LIN {X -0.154,Y -307.907,Z 608.339,A 0.000,B 0.000,C 90.000,E1 61.051} C_DIS
LIN {X 0.052,Y -298.895,Z 608.321,A 0.000,B 0.000,C 90.000,E1 57.740} C_DIS
LIN {X 0.110,Y -290.449,Z 608.302,A 0.000,B 0.000,C 90.000,E1 54.402} C_DIS
LIN {X -0.081,Y -283.937,Z 608.287,A 0.000,B 0.000,C 90.000,E1 51.743} C_DIS
LIN {X 0.078,Y -278.963,Z 608.276,A 0.000,B 0.000,C 90.000,E1 49.666} C_DIS
LIN {X -0.073,Y -273.546,Z 608.265,A 0.000,B 0.000,C 90.000,E1 47.634} C_DIS
LIN {X 0.074,Y -269.596,Z 608.257,A 0.000,B 0.000,C 90.000,E1 46.215} C_DIS
LIN {X -0.146,Y -264.247,Z 608.247,A 0.000,B 0.000,C 90.000,E1 44.514} C_DIS
LIN {X -0.046,Y -257.475,Z 608.235,A 0.000,B 0.000,C 90.000,E1 42.366} C_DIS
LIN {X -0.013,Y -247.381,Z 608.217,A 0.000,B 0.000,C 90.000,E1 39.116} C_DIS
LIN {X 0.041,Y -238.999,Z 608.201,A 0.000,B 0.000,C 90.000,E1 36.171} C_DIS
LIN {X -0.054,Y -231.454,Z 608.184,A 0.000,B 0.000,C 90.000,E1 33.214} C_DIS
LIN {X -0.001,Y -222.964,Z 608.163,A 0.000,B 0.000,C 90.000,E1 29.411} C_DIS
LIN {X -0.110,Y -217.013,Z 608.146,A 0.000,B 0.000,C 90.000,E1 26.360} C_DIS
LIN {X 0.028,Y -211.815,Z 608.129,A 0.000,B 0.000,C 90.000,E1 23.206} C_DIS
LIN {X 0.001,Y -206.428,Z 608.107,A 0.000,B 0.000,C 90.000,E1 19.268} C_DIS
LIN {X -0.072,Y -202.159,Z 608.085,A 0.000,B 0.000,C 90.000,E1 15.300} C_DIS
LIN {X 0.049,Y -198.456,Z 608.058,A 0.000,B 0.000,C 90.000,E1 10.433} C_DIS
LIN {X -0.013,Y -195.902,Z 608.022,A 0.000,B 0.000,C 90.000,E1 3.955} C_DIS
LIN {X 0.064,Y -197.486,Z 607.961,A 0.000,B 0.000,C 90.000,E1 352.996} C_DIS
LIN {X -0.083,Y -200.607,Z 607.934,A 0.000,B 0.000,C 90.000,E1 348.173} C_DIS
LIN {X -0.002,Y -204.996,Z 607.907,A 0.000,B 0.000,C 90.000,E1 343.323} C_DIS
LIN {X -0.001,Y -209.680,Z 607.885,A 0.000,B 0.000,C 90.000,E1 339.337} C_DIS
LIN {X -0.064,Y -215.034,Z 607.863,A 0.000,B 0.000,C 90.000,E1 335.409} C_DIS
LIN {X -0.075,Y -221.104,Z 607.842,A 0.000,B 0.000,C 90.000,E1 331.513} C_DIS
LIN {X -0.057,Y -227.879,Z 607.820,A 0.000,B 0.000,C 90.000,E1 327.661} C_DIS
LIN {X -0.004,Y -233.659,Z 607.803,A 0.000,B 0.000,C 90.000,E1 324.609} C_DIS
LIN {X -0.099,Y -241.291,Z 607.783,A 0.000,B 0.000,C 90.000,E1 320.884} C_DIS
LIN {X 0.101,Y -249.514,Z 607.762,A 0.000,B 0.000,C 90.000,E1 317.148} C_DIS
LIN {X 0.010,Y -258.785,Z 607.742,A 0.000,B 0.000,C 90.000,E1 313.542} C_DIS
LIN {X 0.036,Y -268.335,Z 607.724,A 0.000,B 0.000,C 90.000,E1 310.334} C_DIS
LIN {X -0.067,Y -280.538,Z 607.705,A 0.000,B 0.000,C 90.000,E1 306.870} C_DIS
LIN {X 0.015,Y -292.771,Z 607.688,A 0.000,B 0.000,C 90.000,E1 303.785} C_DIS
LIN {X 0.005,Y -308.160,Z 607.669,A 0.000,B 0.000,C 90.000,E1 300.463} C_DIS
LIN {X 0.131,Y -321.249,Z 607.655,A 0.000,B 0.000,C 90.000,E1 297.847} C_DIS
LIN {X -0.022,Y -336.716,Z 607.639,A 0.000,B 0.000,C 90.000,E1 295.027} C_DIS
LIN {X -0.066,Y -351.631,Z 607.625,A 0.000,B 0.000,C 90.000,E1 292.567} C_DIS
LIN {X -0.076,Y -369.880,Z 607.610,A 0.000,B 0.000,C 90.000,E1 289.866} C_DIS
LIN {X -0.071,Y -385.394,Z 607.599,A 0.000,B 0.000,C 90.000,E1 287.819} C_DIS
LIN {X 0.169,Y -401.771,Z 607.588,A 0.000,B 0.000,C 90.000,E1 285.788} C_DIS
LIN {X 0.044,Y -413.277,Z 607.580,A 0.000,B 0.000,C 90.000,E1 284.411} C_DIS
LIN {X 0.028,Y -426.894,Z 607.571,A 0.000,B 0.000,C 90.000,E1 282.771} C_DIS
LIN {X -0.124,Y -435.553,Z 607.565,A 0.000,B 0.000,C 90.000,E1 281.715} C_DIS
LIN {X 0.033,Y -445.944,Z 607.558,A 0.000,B 0.000,C 90.000,E1 280.366} C_DIS
LIN {X 0.016,Y -453.769,Z 607.552,A 0.000,B 0.000,C 90.000,E1 279.321} C_DIS
LIN {X 0.090,Y -461.171,Z 607.546,A 0.000,B 0.000,C 90.000,E1 278.276} C_DIS
LIN {X 0.189,Y -468.053,Z 607.540,A 0.000,B 0.000,C 90.000,E1 277.239} C_DIS
LIN {X 0.116,Y -472.817,Z 607.536,A 0.000,B 0.000,C 90.000,E1 276.486} C_DIS
LIN {X 0.025,Y -476.986,Z 607.532,A 0.000,B 0.000,C 90.000,E1 275.739} C_DIS
LIN {X 0.162,Y -479.355,Z 607.529,A 0.000,B 0.000,C 90.000,E1 275.220} C_DIS
LIN {X -0.167,Y -481.369,Z 607.526,A 0.000,B 0.000,C 90.000,E1 274.759} C_DIS
LIN {X -0.049,Y -483.017,Z 607.524,A 0.000,B 0.000,C 90.000,E1 274.245} C_DIS
LIN {X 0.120,Y -484.265,Z 607.521,A 0.000,B 0.000,C 90.000,E1 273.726} C_DIS
LIN {X -0.218,Y -485.178,Z 607.518,A 0.000,B 0.000,C 90.000,E1 273.269} C_DIS
LIN {X -0.035,Y -485.791,Z 607.515,A 0.000,B 0.000,C 90.000,E1 272.751} C_DIS
LIN {X 0.127,Y -486.145,Z 607.513,A 0.000,B 0.000,C 90.000,E1 272.236} C_DIS
LIN {X -0.174,Y -486.217,Z 607.510,A 0.000,B 0.000,C 90.000,E1 271.776} C_DIS
LIN {X -0.004,Y -485.806,Z 607.507,A 0.000,B 0.000,C 90.000,E1 271.260} C_DIS
LIN {X 0.167,Y -485.043,Z 607.504,A 0.000,B 0.000,C 90.000,E1 270.745} C_DIS
LIN {X -0.148,Y -483.736,Z 607.501,A 0.000,B 0.000,C 90.000,E1 270.286} C_DIS
LIN {X 0.018,Y -481.794,Z 607.499,A 0.000,B 0.000,C 90.000,E1 269.771} C_DIS
LIN {X -0.143,Y -480.602,Z 607.497,A 0.000,B 0.000,C 90.000,E1 269.542} C_DIS
LIN {X 0.004,Y -477.592,Z 607.495,A 0.000,B 0.000,C 90.000,E1 269.026} C_DIS
LIN {X 0.131,Y -473.643,Z 607.492,A 0.000,B 0.000,C 90.000,E1 268.511} C_DIS
LIN {X -0.047,Y -471.299,Z 607.490,A 0.000,B 0.000,C 90.000,E1 268.282} C_DIS
LIN {X -0.218,Y -468.627,Z 607.489,A 0.000,B 0.000,C 90.000,E1 268.051} C_DIS
LIN {X 0.063,Y -465.586,Z 607.488,A 0.000,B 0.000,C 90.000,E1 267.764} C_DIS
LIN {X 0.139,Y -462.587,Z 607.486,A 0.000,B 0.000,C 90.000,E1 267.535} C_DIS
LIN {X 0.212,Y -459.159,Z 607.485,A 0.000,B 0.000,C 90.000,E1 267.306} C_DIS
LIN {X 0.043,Y -452.159,Z 607.483,A 0.000,B 0.000,C 90.000,E1 266.963} C_DIS
LIN {X -0.010,Y -444.654,Z 607.482,A 0.000,B 0.000,C 90.000,E1 266.674} C_DIS
LIN {X -0.009,Y -436.831,Z 607.480,A 0.000,B 0.000,C 90.000,E1 266.445} C_DIS
LIN {X -0.012,Y -428.139,Z 607.479,A 0.000,B 0.000,C 90.000,E1 266.274} C_DIS
LIN {X -0.015,Y -418.707,Z 607.479,A 0.000,B 0.000,C 90.000,E1 266.159} C_DIS
LIN {X 0.035,Y -410.839,Z 607.478,A 0.000,B 0.000,C 90.000,E1 266.102} C_DIS
LIN {X -0.016,Y -180.925,Z 607.478,A 0.000,B 0.000,C 90.000,E1 266.102} C_DIS
LIN {X -0.023,Y -180.899,Z 607.474,A 0.000,B 0.000,C 90.000,E1 265.241} C_DIS
LIN {X -0.073,Y -180.214,Z 607.464,A 0.000,B 0.000,C 90.000,E1 263.571} C_DIS
LIN {X 0.057,Y -179.034,Z 607.445,A 0.000,B 0.000,C 90.000,E1 260.151} C_DIS
LIN {X -0.057,Y -178.690,Z 607.441,A 0.000,B 0.000,C 90.000,E1 259.342} C_DIS
LIN {X 0.054,Y -175.740,Z 607.412,A 0.000,B 0.000,C 90.000,E1 254.212} C_DIS
LIN {X 0.049,Y -171.924,Z 607.384,A 0.000,B 0.000,C 90.000,E1 249.082} C_DIS
LIN {X 0.024,Y -171.296,Z 607.379,A 0.000,B 0.000,C 90.000,E1 248.230} C_DIS
LIN {X 0.069,Y -167.560,Z 607.355,A 0.000,B 0.000,C 90.000,E1 243.896} C_DIS
LIN {X 0.082,Y -166.184,Z 607.345,A 0.000,B 0.000,C 90.000,E1 242.153} C_DIS
LIN {X 0.072,Y -162.954,Z 607.326,A 0.000,B 0.000,C 90.000,E1 238.663} C_DIS
LIN {X -0.104,Y -160.862,Z 607.311,A 0.000,B 0.000,C 90.000,E1 236.087} C_DIS
LIN {X 0.096,Y -157.638,Z 607.292,A 0.000,B 0.000,C 90.000,E1 232.477} C_DIS
LIN {X 0.034,Y -155.675,Z 607.277,A 0.000,B 0.000,C 90.000,E1 229.828} C_DIS
LIN {X 0.086,Y -151.941,Z 607.252,A 0.000,B 0.000,C 90.000,E1 225.324} C_DIS
LIN {X 0.100,Y -150.180,Z 607.237,A 0.000,B 0.000,C 90.000,E1 222.609} C_DIS
LIN {X 0.020,Y -146.954,Z 607.212,A 0.000,B 0.000,C 90.000,E1 218.096} C_DIS
LIN {X 0.008,Y -145.541,Z 607.196,A 0.000,B 0.000,C 90.000,E1 215.358} C_DIS
LIN {X -0.075,Y -142.937,Z 607.171,A 0.000,B 0.000,C 90.000,E1 210.797} C_DIS
LIN {X -0.019,Y -141.561,Z 607.150,A 0.000,B 0.000,C 90.000,E1 207.078} C_DIS
LIN {X 0.034,Y -139.409,Z 607.114,A 0.000,B 0.000,C 90.000,E1 200.556} C_DIS
LIN {X -0.044,Y -139.130,Z 607.104,A 0.000,B 0.000,C 90.000,E1 198.725} C_DIS
LIN {X -0.017,Y -138.350,Z 607.057,A 0.000,B 0.000,C 90.000,E1 190.310} C_DIS
LIN {X -0.029,Y -139.498,Z 607.005,A 0.000,B 0.000,C 90.000,E1 180.974} C_DIS
LIN {X 0.052,Y -141.119,Z 606.974,A 0.000,B 0.000,C 90.000,E1 175.355} C_DIS
LIN {X 0.005,Y -142.499,Z 606.959,A 0.000,B 0.000,C 90.000,E1 172.591} C_DIS
LIN {X -0.048,Y -144.754,Z 606.933,A 0.000,B 0.000,C 90.000,E1 167.993} C_DIS
LIN {X 0.043,Y -147.363,Z 606.913,A 0.000,B 0.000,C 90.000,E1 164.283} C_DIS
LIN {X -0.035,Y -150.690,Z 606.887,A 0.000,B 0.000,C 90.000,E1 159.752} C_DIS
LIN {X 0.048,Y -154.170,Z 606.867,A 0.000,B 0.000,C 90.000,E1 156.102} C_DIS
LIN {X -0.022,Y -157.604,Z 606.847,A 0.000,B 0.000,C 90.000,E1 152.538} C_DIS
LIN {X -0.072,Y -161.856,Z 606.828,A 0.000,B 0.000,C 90.000,E1 148.997} C_DIS
LIN {X -0.054,Y -166.047,Z 606.808,A 0.000,B 0.000,C 90.000,E1 145.468} C_DIS
LIN {X -0.063,Y -171.051,Z 606.789,A 0.000,B 0.000,C 90.000,E1 141.984} C_DIS
LIN {X -0.033,Y -175.922,Z 606.770,A 0.000,B 0.000,C 90.000,E1 138.528} C_DIS
LIN {X -0.041,Y -180.161,Z 606.755,A 0.000,B 0.000,C 90.000,E1 135.972} C_DIS
LIN {X -0.072,Y -185.579,Z 606.737,A 0.000,B 0.000,C 90.000,E1 132.609} C_DIS
LIN {X -0.035,Y -191.262,Z 606.719,A 0.000,B 0.000,C 90.000,E1 129.483} C_DIS
LIN {X -0.093,Y -288.943,Z 606.719,A 0.000,B 0.000,C 90.000,E1 129.483} C_DIS
LIN {X -0.106,Y -294.294,Z 606.718,A 0.000,B 0.000,C 90.000,E1 129.277} C_DIS
LIN {X 0.030,Y -297.356,Z 606.717,A 0.000,B 0.000,C 90.000,E1 128.991} C_DIS
LIN {X -0.045,Y -301.065,Z 606.714,A 0.000,B 0.000,C 90.000,E1 128.508} C_DIS
LIN {X -0.051,Y -302.796,Z 606.712,A 0.000,B 0.000,C 90.000,E1 128.177} C_DIS
LIN {X 0.131,Y -304.154,Z 606.710,A 0.000,B 0.000,C 90.000,E1 127.810} C_DIS
LIN {X 0.085,Y -307.941,Z 606.703,A 0.000,B 0.000,C 90.000,E1 126.503} C_DIS
LIN {X -0.122,Y -317.977,Z 606.685,A 0.000,B 0.000,C 90.000,E1 123.293} C_DIS
LIN {X 0.095,Y -328.326,Z 606.669,A 0.000,B 0.000,C 90.000,E1 120.384} C_DIS
LIN {X -0.045,Y -340.030,Z 606.653,A 0.000,B 0.000,C 90.000,E1 117.590} C_DIS
LIN {X -0.003,Y -353.187,Z 606.638,A 0.000,B 0.000,C 90.000,E1 114.823} C_DIS
LIN {X 0.076,Y -366.203,Z 606.625,A 0.000,B 0.000,C 90.000,E1 112.408} C_DIS
LIN {X 0.018,Y -380.557,Z 606.612,A 0.000,B 0.000,C 90.000,E1 110.066} C_DIS
LIN {X 0.054,Y -396.354,Z 606.599,A 0.000,B 0.000,C 90.000,E1 107.764} C_DIS
LIN {X -0.143,Y -413.709,Z 606.586,A 0.000,B 0.000,C 90.000,E1 105.552} C_DIS
LIN {X -0.022,Y -432.735,Z 606.574,A 0.000,B 0.000,C 90.000,E1 103.355} C_DIS
LIN {X 0.049,Y -452.847,Z 606.563,A 0.000,B 0.000,C 90.000,E1 101.299} C_DIS
LIN {X -0.132,Y -473.327,Z 606.552,A 0.000,B 0.000,C 90.000,E1 99.443} C_DIS
LIN {X -0.043,Y -475.167,Z 606.551,A 0.000,B 0.000,C 90.000,E1 99.208} C_DIS
LIN {X -0.182,Y -476.735,Z 606.550,A 0.000,B 0.000,C 90.000,E1 98.973} C_DIS
LIN {X 0.077,Y -477.911,Z 606.548,A 0.000,B 0.000,C 90.000,E1 98.690} C_DIS
LIN {X -0.186,Y -479.333,Z 606.546,A 0.000,B 0.000,C 90.000,E1 98.219} C_DIS
LIN {X -0.038,Y -479.722,Z 606.543,A 0.000,B 0.000,C 90.000,E1 97.701} C_DIS
LIN {X 0.120,Y -479.141,Z 606.540,A 0.000,B 0.000,C 90.000,E1 97.182} C_DIS
LIN {X -0.194,Y -477.502,Z 606.537,A 0.000,B 0.000,C 90.000,E1 96.720} C_DIS
LIN {X 0.149,Y -476.194,Z 606.536,A 0.000,B 0.000,C 90.000,E1 96.429} C_DIS
LIN {X 0.012,Y -465.298,Z 606.527,A 0.000,B 0.000,C 90.000,E1 94.935} C_DIS
LIN {X 0.163,Y -455.064,Z 606.519,A 0.000,B 0.000,C 90.000,E1 93.383} C_DIS
LIN {X 0.069,Y -442.818,Z 606.507,A 0.000,B 0.000,C 90.000,E1 91.318} C_DIS
LIN {X -0.195,Y -434.234,Z 606.499,A 0.000,B 0.000,C 90.000,E1 89.771} C_DIS
LIN {X 0.119,Y -426.716,Z 606.491,A 0.000,B 0.000,C 90.000,E1 88.396} C_DIS
LIN {X 0.033,Y -417.283,Z 606.482,A 0.000,B 0.000,C 90.000,E1 86.788} C_DIS
LIN {X 0.018,Y -403.197,Z 606.468,A 0.000,B 0.000,C 90.000,E1 84.318} C_DIS
LIN {X 0.155,Y -388.249,Z 606.453,A 0.000,B 0.000,C 90.000,E1 81.489} C_DIS
LIN {X -0.001,Y -376.701,Z 606.440,A 0.000,B 0.000,C 90.000,E1 79.218} C_DIS
LIN {X 0.012,Y -365.513,Z 606.427,A 0.000,B 0.000,C 90.000,E1 76.881} C_DIS
LIN {X -0.100,Y -352.191,Z 606.411,A 0.000,B 0.000,C 90.000,E1 73.921} C_DIS
LIN {X 0.021,Y -337.507,Z 606.390,A 0.000,B 0.000,C 90.000,E1 70.242} C_DIS
LIN {X 0.131,Y -325.514,Z 606.371,A 0.000,B 0.000,C 90.000,E1 66.794} C_DIS
LIN {X 0.015,Y -315.551,Z 606.354,A 0.000,B 0.000,C 90.000,E1 63.640} C_DIS
LIN {X 0.068,Y -308.120,Z 606.339,A 0.000,B 0.000,C 90.000,E1 61.051} C_DIS
LIN {X 0.021,Y -299.091,Z 606.321,A 0.000,B 0.000,C 90.000,E1 57.788} C_DIS
LIN {X -0.074,Y -290.637,Z 606.303,A 0.000,B 0.000,C 90.000,E1 54.482} C_DIS
LIN {X -0.036,Y -284.120,Z 606.288,A 0.000,B 0.000,C 90.000,E1 51.778} C_DIS
LIN {X -0.095,Y -279.147,Z 606.276,A 0.000,B 0.000,C 90.000,E1 49.747} C_DIS
LIN {X -0.056,Y -273.737,Z 606.265,A 0.000,B 0.000,C 90.000,E1 47.676} C_DIS
LIN {X -0.089,Y -269.777,Z 606.257,A 0.000,B 0.000,C 90.000,E1 46.296} C_DIS
LIN {X 0.009,Y -265.547,Z 606.249,A 0.000,B 0.000,C 90.000,E1 44.879} C_DIS
LIN {X -0.041,Y -258.820,Z 606.238,A 0.000,B 0.000,C 90.000,E1 42.771} C_DIS
LIN {X 0.015,Y -249.763,Z 606.222,A 0.000,B 0.000,C 90.000,E1 39.886} C_DIS
LIN {X 0.063,Y -239.141,Z 606.201,A 0.000,B 0.000,C 90.000,E1 36.217} C_DIS
LIN {X 0.031,Y -231.589,Z 606.185,A 0.000,B 0.000,C 90.000,E1 33.245} C_DIS
LIN {X 0.080,Y -224.692,Z 606.168,A 0.000,B 0.000,C 90.000,E1 30.207} C_DIS
LIN {X 0.115,Y -218.544,Z 606.151,A 0.000,B 0.000,C 90.000,E1 27.129} C_DIS
LIN {X -0.103,Y -213.122,Z 606.134,A 0.000,B 0.000,C 90.000,E1 24.079} C_DIS
LIN {X -0.011,Y -207.491,Z 606.112,A 0.000,B 0.000,C 90.000,E1 20.120} C_DIS
LIN {X 0.009,Y -202.956,Z 606.090,A 0.000,B 0.000,C 90.000,E1 16.134} C_DIS
LIN {X 0.047,Y -199.020,Z 606.063,A 0.000,B 0.000,C 90.000,E1 11.299} C_DIS
LIN {X 0.036,Y -196.308,Z 606.031,A 0.000,B 0.000,C 90.000,E1 5.625} C_DIS
LIN {X 0.064,Y -197.506,Z 605.961,A 0.000,B 0.000,C 90.000,E1 352.996} C_DIS
LIN {X -0.081,Y -200.649,Z 605.934,A 0.000,B 0.000,C 90.000,E1 348.173} C_DIS
LIN {X 0.000,Y -205.029,Z 605.907,A 0.000,B 0.000,C 90.000,E1 343.323} C_DIS
LIN {X 0.003,Y -209.708,Z 605.885,A 0.000,B 0.000,C 90.000,E1 339.337} C_DIS
LIN {X -0.059,Y -215.060,Z 605.863,A 0.000,B 0.000,C 90.000,E1 335.409} C_DIS
LIN {X -0.068,Y -221.137,Z 605.842,A 0.000,B 0.000,C 90.000,E1 331.513} C_DIS
LIN {X -0.050,Y -227.896,Z 605.820,A 0.000,B 0.000,C 90.000,E1 327.661} C_DIS
LIN {X -0.030,Y -235.138,Z 605.799,A 0.000,B 0.000,C 90.000,E1 323.863} C_DIS
LIN {X 0.025,Y -242.853,Z 605.778,A 0.000,B 0.000,C 90.000,E1 320.114} C_DIS
LIN {X -0.070,Y -251.235,Z 605.758,A 0.000,B 0.000,C 90.000,E1 316.458} C_DIS
LIN {X -0.111,Y -260.744,Z 605.738,A 0.000,B 0.000,C 90.000,E1 312.852} C_DIS
LIN {X -0.023,Y -270.590,Z 605.720,A 0.000,B 0.000,C 90.000,E1 309.644} C_DIS
LIN {X -0.007,Y -283.114,Z 605.701,A 0.000,B 0.000,C 90.000,E1 306.171} C_DIS
LIN {X 0.019,Y -292.723,Z 605.688,A 0.000,B 0.000,C 90.000,E1 303.785} C_DIS
LIN {X 0.005,Y -308.088,Z 605.669,A 0.000,B 0.000,C 90.000,E1 300.463} C_DIS
LIN {X 0.129,Y -321.151,Z 605.655,A 0.000,B 0.000,C 90.000,E1 297.847} C_DIS
LIN {X -0.051,Y -338.391,Z 605.637,A 0.000,B 0.000,C 90.000,E1 294.719} C_DIS
LIN {X -0.016,Y -355.459,Z 605.622,A 0.000,B 0.000,C 90.000,E1 291.950} C_DIS
LIN {X -0.126,Y -371.969,Z 605.609,A 0.000,B 0.000,C 90.000,E1 289.577} C_DIS
LIN {X -0.076,Y -397.069,Z 605.591,A 0.000,B 0.000,C 90.000,E1 286.386} C_DIS
LIN {X 0.121,Y -408.725,Z 605.583,A 0.000,B 0.000,C 90.000,E1 284.954} C_DIS
LIN {X -0.135,Y -424.690,Z 605.572,A 0.000,B 0.000,C 90.000,E1 283.063} C_DIS
LIN {X 0.106,Y -433.465,Z 605.566,A 0.000,B 0.000,C 90.000,E1 281.951} C_DIS
LIN {X -0.189,Y -443.962,Z 605.559,A 0.000,B 0.000,C 90.000,E1 280.658} C_DIS
LIN {X 0.213,Y -451.909,Z 605.553,A 0.000,B 0.000,C 90.000,E1 279.557} C_DIS
LIN {X -0.183,Y -459.380,Z 605.547,A 0.000,B 0.000,C 90.000,E1 278.568} C_DIS
LIN {X -0.109,Y -466.347,Z 605.542,A 0.000,B 0.000,C 90.000,E1 277.530} C_DIS
LIN {X 0.111,Y -472.755,Z 605.536,A 0.000,B 0.000,C 90.000,E1 276.486} C_DIS
LIN {X 0.019,Y -476.899,Z 605.532,A 0.000,B 0.000,C 90.000,E1 275.739} C_DIS
LIN {X 0.155,Y -479.288,Z 605.529,A 0.000,B 0.000,C 90.000,E1 275.220} C_DIS
LIN {X -0.174,Y -481.306,Z 605.526,A 0.000,B 0.000,C 90.000,E1 274.759} C_DIS
LIN {X -0.056,Y -482.966,Z 605.524,A 0.000,B 0.000,C 90.000,E1 274.245} C_DIS
LIN {X 0.112,Y -484.232,Z 605.521,A 0.000,B 0.000,C 90.000,E1 273.726} C_DIS
LIN {X -0.225,Y -485.166,Z 605.518,A 0.000,B 0.000,C 90.000,E1 273.269} C_DIS
LIN {X -0.044,Y -485.815,Z 605.515,A 0.000,B 0.000,C 90.000,E1 272.751} C_DIS
LIN {X 0.120,Y -486.126,Z 605.513,A 0.000,B 0.000,C 90.000,E1 272.236} C_DIS
LIN {X -0.182,Y -486.172,Z 605.510,A 0.000,B 0.000,C 90.000,E1 271.776} C_DIS
LIN {X -0.013,Y -485.880,Z 605.507,A 0.000,B 0.000,C 90.000,E1 271.260} C_DIS
LIN {X 0.159,Y -485.075,Z 605.504,A 0.000,B 0.000,C 90.000,E1 270.745} C_DIS
LIN {X -0.156,Y -483.746,Z 605.501,A 0.000,B 0.000,C 90.000,E1 270.286} C_DIS
LIN {X 0.010,Y -481.874,Z 605.499,A 0.000,B 0.000,C 90.000,E1 269.771} C_DIS
LIN {X 0.167,Y -479.239,Z 605.496,A 0.000,B 0.000,C 90.000,E1 269.255} C_DIS
LIN {X -0.173,Y -475.770,Z 605.493,A 0.000,B 0.000,C 90.000,E1 268.797} C_DIS
LIN {X -0.054,Y -471.288,Z 605.490,A 0.000,B 0.000,C 90.000,E1 268.282} C_DIS
LIN {X -0.225,Y -468.587,Z 605.489,A 0.000,B 0.000,C 90.000,E1 268.051} C_DIS
LIN {X 0.056,Y -465.563,Z 605.488,A 0.000,B 0.000,C 90.000,E1 267.764} C_DIS
LIN {X 0.125,Y -462.549,Z 605.486,A 0.000,B 0.000,C 90.000,E1 267.535} C_DIS
LIN {X 0.192,Y -459.093,Z 605.485,A 0.000,B 0.000,C 90.000,E1 267.306} C_DIS
LIN {X 0.031,Y -452.126,Z 605.483,A 0.000,B 0.000,C 90.000,E1 266.963} C_DIS
LIN {X -0.034,Y -444.549,Z 605.482,A 0.000,B 0.000,C 90.000,E1 266.674} C_DIS
LIN {X -0.010,Y -436.839,Z 605.480,A 0.000,B 0.000,C 90.000,E1 266.445} C_DIS
LIN {X 0.003,Y -428.221,Z 605.479,A 0.000,B 0.000,C 90.000,E1 266.274} C_DIS
LIN {X 0.001,Y -418.631,Z 605.479,A 0.000,B 0.000,C 90.000,E1 266.159} C_DIS
LIN {X 0.053,Y -411.194,Z 605.478,A 0.000,B 0.000,C 90.000,E1 266.102} C_DIS
LIN {X -0.020,Y -405.738,Z 605.478,A 0.000,B 0.000,C 90.000,E1 266.102} C_DIS
LIN {X -0.040,Y -180.924,Z 605.478,A 0.000,B 0.000,C 90.000,E1 266.102} C_DIS
LIN {X 0.004,Y -180.875,Z 605.473,A 0.000,B 0.000,C 90.000,E1 265.065} C_DIS
LIN {X 0.087,Y -178.942,Z 605.443,A 0.000,B 0.000,C 90.000,E1 259.803} C_DIS
LIN {X -0.046,Y -175.992,Z 605.415,A 0.000,B 0.000,C 90.000,E1 254.755} C_DIS
LIN {X 0.069,Y -175.495,Z 605.410,A 0.000,B 0.000,C 90.000,E1 253.866} C_DIS
LIN {X -0.037,Y -172.238,Z 605.387,A 0.000,B 0.000,C 90.000,E1 249.625} C_DIS
LIN {X -0.058,Y -171.715,Z 605.382,A 0.000,B 0.000,C 90.000,E1 248.773} C_DIS
LIN {X 0.026,Y -167.311,Z 605.353,A 0.000,B 0.000,C 90.000,E1 243.563} C_DIS
LIN {X 0.032,Y -166.691,Z 605.348,A 0.000,B 0.000,C 90.000,E1 242.692} C_DIS
LIN {X 0.023,Y -162.673,Z 605.324,A 0.000,B 0.000,C 90.000,E1 238.329} C_DIS
LIN {X -0.004,Y -161.362,Z 605.314,A 0.000,B 0.000,C 90.000,E1 236.580} C_DIS
LIN {X 0.030,Y -157.356,Z 605.290,A 0.000,B 0.000,C 90.000,E1 232.145} C_DIS
LIN {X 0.058,Y -155.345,Z 605.275,A 0.000,B 0.000,C 90.000,E1 229.461} C_DIS
LIN {X -0.012,Y -151.692,Z 605.250,A 0.000,B 0.000,C 90.000,E1 225.000} C_DIS
LIN {X 0.036,Y -150.554,Z 605.240,A 0.000,B 0.000,C 90.000,E1 223.176} C_DIS
LIN {X -0.047,Y -147.281,Z 605.215,A 0.000,B 0.000,C 90.000,E1 218.669} C_DIS
LIN {X 0.040,Y -145.309,Z 605.194,A 0.000,B 0.000,C 90.000,E1 214.978} C_DIS
LIN {X 0.032,Y -142.399,Z 605.164,A 0.000,B 0.000,C 90.000,E1 209.461} C_DIS
LIN {X 0.015,Y -141.382,Z 605.148,A 0.000,B 0.000,C 90.000,E1 206.693} C_DIS
LIN {X 0.056,Y -139.349,Z 605.112,A 0.000,B 0.000,C 90.000,E1 200.174} C_DIS
LIN {X -0.002,Y -138.787,Z 605.097,A 0.000,B 0.000,C 90.000,E1 197.402} C_DIS
LIN {X 0.056,Y -138.344,Z 605.055,A 0.000,B 0.000,C 90.000,E1 189.905} C_DIS
LIN {X -0.063,Y -139.386,Z 605.008,A 0.000,B 0.000,C 90.000,E1 181.547} C_DIS
LIN {X -0.010,Y -141.283,Z 604.972,A 0.000,B 0.000,C 90.000,E1 175.008} C_DIS
LIN {X -0.052,Y -142.646,Z 604.957,A 0.000,B 0.000,C 90.000,E1 172.243} C_DIS
LIN {X 0.039,Y -144.982,Z 604.931,A 0.000,B 0.000,C 90.000,E1 167.589} C_DIS
LIN {X 0.030,Y -147.610,Z 604.911,A 0.000,B 0.000,C 90.000,E1 163.921} C_DIS
LIN {X -0.032,Y -150.232,Z 604.890,A 0.000,B 0.000,C 90.000,E1 160.296} C_DIS
LIN {X -0.017,Y -153.623,Z 604.870,A 0.000,B 0.000,C 90.000,E1 156.666} C_DIS
LIN {X -0.029,Y -157.040,Z 604.850,A 0.000,B 0.000,C 90.000,E1 153.076} C_DIS
LIN {X 0.040,Y -161.165,Z 604.831,A 0.000,B 0.000,C 90.000,E1 149.488} C_DIS
LIN {X -0.016,Y -163.261,Z 604.821,A 0.000,B 0.000,C 90.000,E1 147.740} C_DIS
LIN {X 0.082,Y -167.699,Z 604.801,A 0.000,B 0.000,C 90.000,E1 144.196} C_DIS
LIN {X -0.005,Y -171.520,Z 604.787,A 0.000,B 0.000,C 90.000,E1 141.618} C_DIS
LIN {X 0.038,Y -176.458,Z 604.768,A 0.000,B 0.000,C 90.000,E1 138.162} C_DIS
LIN {X -0.091,Y -180.754,Z 604.753,A 0.000,B 0.000,C 90.000,E1 135.648} C_DIS
LIN {X 0.027,Y -186.159,Z 604.735,A 0.000,B 0.000,C 90.000,E1 132.243} C_DIS
LIN {X -0.052,Y -191.271,Z 604.719,A 0.000,B 0.000,C 90.000,E1 129.483} C_DIS
LIN {X -0.114,Y -288.437,Z 604.719,A 0.000,B 0.000,C 90.000,E1 129.483} C_DIS
LIN {X 0.031,Y -291.041,Z 604.719,A 0.000,B 0.000,C 90.000,E1 129.402} C_DIS
LIN {X -0.154,Y -295.400,Z 604.718,A 0.000,B 0.000,C 90.000,E1 129.197} C_DIS
LIN {X 0.078,Y -297.932,Z 604.716,A 0.000,B 0.000,C 90.000,E1 128.910} C_DIS
LIN {X -0.022,Y -301.701,Z 604.713,A 0.000,B 0.000,C 90.000,E1 128.382} C_DIS
LIN {X 0.161,Y -303.293,Z 604.711,A 0.000,B 0.000,C 90.000,E1 128.016} C_DIS
LIN {X -0.081,Y -304.544,Z 604.710,A 0.000,B 0.000,C 90.000,E1 127.729} C_DIS
LIN {X 0.066,Y -316.213,Z 604.688,A 0.000,B 0.000,C 90.000,E1 123.785} C_DIS
LIN {X -0.035,Y -326.327,Z 604.672,A 0.000,B 0.000,C 90.000,E1 120.924} C_DIS
LIN {X -0.072,Y -337.778,Z 604.656,A 0.000,B 0.000,C 90.000,E1 118.103} C_DIS
LIN {X -0.098,Y -350.662,Z 604.641,A 0.000,B 0.000,C 90.000,E1 115.335} C_DIS
LIN {X 0.058,Y -363.416,Z 604.627,A 0.000,B 0.000,C 90.000,E1 112.898} C_DIS
LIN {X -0.075,Y -377.489,Z 604.614,A 0.000,B 0.000,C 90.000,E1 110.556} C_DIS
LIN {X 0.005,Y -392.981,Z 604.601,A 0.000,B 0.000,C 90.000,E1 108.236} C_DIS
LIN {X 0.110,Y -410.008,Z 604.589,A 0.000,B 0.000,C 90.000,E1 105.969} C_DIS
LIN {X 0.141,Y -428.692,Z 604.577,A 0.000,B 0.000,C 90.000,E1 103.772} C_DIS
LIN {X -0.049,Y -448.669,Z 604.565,A 0.000,B 0.000,C 90.000,E1 101.715} C_DIS
LIN {X 0.043,Y -469.223,Z 604.554,A 0.000,B 0.000,C 90.000,E1 99.792} C_DIS
LIN {X 0.100,Y -471.843,Z 604.553,A 0.000,B 0.000,C 90.000,E1 99.557} C_DIS
LIN {X 0.196,Y -474.068,Z 604.552,A 0.000,B 0.000,C 90.000,E1 99.321} C_DIS
LIN {X -0.253,Y -475.755,Z 604.551,A 0.000,B 0.000,C 90.000,E1 99.151} C_DIS
LIN {X 0.080,Y -477.205,Z 604.549,A 0.000,B 0.000,C 90.000,E1 98.859} C_DIS
LIN {X -0.057,Y -478.285,Z 604.548,A 0.000,B 0.000,C 90.000,E1 98.624} C_DIS
LIN {X 0.086,Y -479.555,Z 604.545,A 0.000,B 0.000,C 90.000,E1 98.106} C_DIS
LIN {X -0.238,Y -479.811,Z 604.542,A 0.000,B 0.000,C 90.000,E1 97.644} C_DIS
LIN {X -0.078,Y -479.095,Z 604.540,A 0.000,B 0.000,C 90.000,E1 97.125} C_DIS
LIN {X 0.083,Y -477.291,Z 604.537,A 0.000,B 0.000,C 90.000,E1 96.606} C_DIS
LIN {X -0.048,Y -475.875,Z 604.535,A 0.000,B 0.000,C 90.000,E1 96.372} C_DIS
LIN {X 0.146,Y -459.619,Z 604.523,A 0.000,B 0.000,C 90.000,E1 94.073} C_DIS
LIN {X 0.162,Y -446.885,Z 604.511,A 0.000,B 0.000,C 90.000,E1 92.007} C_DIS
LIN {X -0.125,Y -435.320,Z 604.500,A 0.000,B 0.000,C 90.000,E1 89.943} C_DIS
LIN {X 0.202,Y -427.861,Z 604.492,A 0.000,B 0.000,C 90.000,E1 88.568} C_DIS
LIN {X 0.111,Y -418.438,Z 604.483,A 0.000,B 0.000,C 90.000,E1 86.963} C_DIS
LIN {X 0.154,Y -404.322,Z 604.469,A 0.000,B 0.000,C 90.000,E1 84.489} C_DIS
LIN {X -0.115,Y -389.328,Z 604.454,A 0.000,B 0.000,C 90.000,E1 81.724} C_DIS
LIN {X 0.144,Y -376.306,Z 604.440,A 0.000,B 0.000,C 90.000,E1 79.106} C_DIS
LIN {X 0.137,Y -365.118,Z 604.427,A 0.000,B 0.000,C 90.000,E1 76.769} C_DIS
LIN {X 0.035,Y -350.543,Z 604.408,A 0.000,B 0.000,C 90.000,E1 73.504} C_DIS
LIN {X 0.087,Y -336.050,Z 604.388,A 0.000,B 0.000,C 90.000,E1 69.826} C_DIS
LIN {X -0.074,Y -323.207,Z 604.367,A 0.000,B 0.000,C 90.000,E1 66.102} C_DIS
LIN {X 0.168,Y -313.460,Z 604.349,A 0.000,B 0.000,C 90.000,E1 62.871} C_DIS
LIN {X -0.105,Y -306.068,Z 604.335,A 0.000,B 0.000,C 90.000,E1 60.333} C_DIS
LIN {X -0.056,Y -297.174,Z 604.317,A 0.000,B 0.000,C 90.000,E1 57.041} C_DIS
LIN {X 0.050,Y -290.463,Z 604.302,A 0.000,B 0.000,C 90.000,E1 54.356} C_DIS
LIN {X 0.028,Y -283.942,Z 604.287,A 0.000,B 0.000,C 90.000,E1 51.662} C_DIS
LIN {X 0.006,Y -278.952,Z 604.276,A 0.000,B 0.000,C 90.000,E1 49.622} C_DIS
LIN {X 0.035,Y -275.379,Z 604.268,A 0.000,B 0.000,C 90.000,E1 48.243} C_DIS
LIN {X 0.019,Y -271.537,Z 604.260,A 0.000,B 0.000,C 90.000,E1 46.863} C_DIS
LIN {X -0.053,Y -267.416,Z 604.253,A 0.000,B 0.000,C 90.000,E1 45.486} C_DIS
LIN {X 0.064,Y -261.905,Z 604.243,A 0.000,B 0.000,C 90.000,E1 43.704} C_DIS
LIN {X 0.001,Y -252.812,Z 604.227,A 0.000,B 0.000,C 90.000,E1 40.862} C_DIS
LIN {X -0.052,Y -242.975,Z 604.209,A 0.000,B 0.000,C 90.000,E1 37.604} C_DIS
LIN {X 0.093,Y -234.981,Z 604.192,A 0.000,B 0.000,C 90.000,E1 34.612} C_DIS
LIN {X -0.013,Y -226.101,Z 604.172,A 0.000,B 0.000,C 90.000,E1 30.875} C_DIS
LIN {X -0.132,Y -219.775,Z 604.155,A 0.000,B 0.000,C 90.000,E1 27.847} C_DIS
LIN {X -0.025,Y -214.201,Z 604.137,A 0.000,B 0.000,C 90.000,E1 24.719} C_DIS
LIN {X -0.045,Y -209.443,Z 604.120,A 0.000,B 0.000,C 90.000,E1 21.589} C_DIS
LIN {X -0.091,Y -204.485,Z 604.098,A 0.000,B 0.000,C 90.000,E1 17.638} C_DIS
LIN {X 0.055,Y -200.708,Z 604.076,A 0.000,B 0.000,C 90.000,E1 13.592} C_DIS
LIN {X 0.049,Y -197.487,Z 604.049,A 0.000,B 0.000,C 90.000,E1 8.746} C_DIS
LIN {X 0.049,Y -198.424,Z 603.952,A 0.000,B 0.000,C 90.000,E1 351.376} C_DIS
LIN {X 0.013,Y -202.029,Z 603.925,A 0.000,B 0.000,C 90.000,E1 346.533} C_DIS
LIN {X -0.070,Y -205.948,Z 603.903,A 0.000,B 0.000,C 90.000,E1 342.543} C_DIS
LIN {X 0.028,Y -210.754,Z 603.881,A 0.000,B 0.000,C 90.000,E1 338.539} C_DIS
LIN {X 0.087,Y -216.241,Z 603.859,A 0.000,B 0.000,C 90.000,E1 334.588} C_DIS
LIN {X 0.025,Y -222.452,Z 603.837,A 0.000,B 0.000,C 90.000,E1 330.717} C_DIS
LIN {X -0.107,Y -229.330,Z 603.816,A 0.000,B 0.000,C 90.000,E1 326.914} C_DIS
LIN {X -0.100,Y -236.619,Z 603.795,A 0.000,B 0.000,C 90.000,E1 323.130} C_DIS
LIN {X 0.006,Y -244.429,Z 603.774,A 0.000,B 0.000,C 90.000,E1 319.380} C_DIS
LIN {X -0.058,Y -252.996,Z 603.754,A 0.000,B 0.000,C 90.000,E1 315.729} C_DIS
LIN {X -0.037,Y -262.758,Z 603.734,A 0.000,B 0.000,C 90.000,E1 312.123} C_DIS
LIN {X 0.057,Y -271.704,Z 603.718,A 0.000,B 0.000,C 90.000,E1 309.277} C_DIS
LIN {X 0.115,Y -284.386,Z 603.699,A 0.000,B 0.000,C 90.000,E1 305.804} C_DIS
LIN {X 0.008,Y -294.128,Z 603.686,A 0.000,B 0.000,C 90.000,E1 303.452} C_DIS
LIN {X 0.043,Y -309.612,Z 603.667,A 0.000,B 0.000,C 90.000,E1 300.129} C_DIS
LIN {X -0.152,Y -324.412,Z 603.651,A 0.000,B 0.000,C 90.000,E1 297.257} C_DIS
LIN {X 0.059,Y -341.947,Z 603.634,A 0.000,B 0.000,C 90.000,E1 294.079} C_DIS
LIN {X -0.072,Y -359.392,Z 603.619,A 0.000,B 0.000,C 90.000,E1 291.354} C_DIS
LIN {X -0.049,Y -374.104,Z 603.607,A 0.000,B 0.000,C 90.000,E1 289.268} C_DIS
LIN {X -0.089,Y -397.084,Z 603.591,A 0.000,B 0.000,C 90.000,E1 286.386} C_DIS
LIN {X 0.108,Y -408.699,Z 603.583,A 0.000,B 0.000,C 90.000,E1 284.954} C_DIS
LIN {X 0.112,Y -422.447,Z 603.574,A 0.000,B 0.000,C 90.000,E1 283.300} C_DIS
LIN {X -0.090,Y -431.352,Z 603.568,A 0.000,B 0.000,C 90.000,E1 282.243} C_DIS
LIN {X 0.008,Y -441.994,Z 603.561,A 0.000,B 0.000,C 90.000,E1 280.894} C_DIS
LIN {X -0.054,Y -450.044,Z 603.555,A 0.000,B 0.000,C 90.000,E1 279.849} C_DIS
LIN {X -0.205,Y -459.418,Z 603.547,A 0.000,B 0.000,C 90.000,E1 278.568} C_DIS
LIN {X -0.129,Y -466.350,Z 603.542,A 0.000,B 0.000,C 90.000,E1 277.530} C_DIS
LIN {X 0.089,Y -472.720,Z 603.536,A 0.000,B 0.000,C 90.000,E1 276.486} C_DIS
LIN {X -0.003,Y -476.856,Z 603.532,A 0.000,B 0.000,C 90.000,E1 275.739} C_DIS
LIN {X -0.052,Y -480.281,Z 603.528,A 0.000,B 0.000,C 90.000,E1 274.992} C_DIS
LIN {X -0.197,Y -481.280,Z 603.526,A 0.000,B 0.000,C 90.000,E1 274.759} C_DIS
LIN {X -0.073,Y -482.929,Z 603.524,A 0.000,B 0.000,C 90.000,E1 274.245} C_DIS
LIN {X 0.095,Y -484.197,Z 603.521,A 0.000,B 0.000,C 90.000,E1 273.726} C_DIS
LIN {X -0.243,Y -485.141,Z 603.518,A 0.000,B 0.000,C 90.000,E1 273.269} C_DIS
LIN {X -0.062,Y -485.826,Z 603.515,A 0.000,B 0.000,C 90.000,E1 272.751} C_DIS
LIN {X 0.101,Y -486.168,Z 603.513,A 0.000,B 0.000,C 90.000,E1 272.236} C_DIS
LIN {X -0.200,Y -486.232,Z 603.510,A 0.000,B 0.000,C 90.000,E1 271.776} C_DIS
LIN {X -0.030,Y -485.939,Z 603.507,A 0.000,B 0.000,C 90.000,E1 271.260} C_DIS
LIN {X 0.142,Y -485.116,Z 603.504,A 0.000,B 0.000,C 90.000,E1 270.745} C_DIS
LIN {X -0.172,Y -483.814,Z 603.501,A 0.000,B 0.000,C 90.000,E1 270.286} C_DIS
LIN {X -0.006,Y -481.893,Z 603.499,A 0.000,B 0.000,C 90.000,E1 269.771} C_DIS
LIN {X 0.151,Y -479.265,Z 603.496,A 0.000,B 0.000,C 90.000,E1 269.255} C_DIS
LIN {X -0.189,Y -475.785,Z 603.493,A 0.000,B 0.000,C 90.000,E1 268.797} C_DIS
LIN {X 0.108,Y -473.674,Z 603.492,A 0.000,B 0.000,C 90.000,E1 268.511} C_DIS
LIN {X 0.232,Y -468.586,Z 603.489,A 0.000,B 0.000,C 90.000,E1 267.993} C_DIS
LIN {X 0.049,Y -465.556,Z 603.488,A 0.000,B 0.000,C 90.000,E1 267.764} C_DIS
LIN {X 0.194,Y -459.106,Z 603.485,A 0.000,B 0.000,C 90.000,E1 267.306} C_DIS
LIN {X 0.003,Y -452.041,Z 603.483,A 0.000,B 0.000,C 90.000,E1 266.963} C_DIS
LIN {X -0.066,Y -444.444,Z 603.481,A 0.000,B 0.000,C 90.000,E1 266.674} C_DIS
LIN {X -0.038,Y -436.727,Z 603.480,A 0.000,B 0.000,C 90.000,E1 266.445} C_DIS
LIN {X -0.017,Y -428.020,Z 603.479,A 0.000,B 0.000,C 90.000,E1 266.274} C_DIS
LIN {X -0.005,Y -418.362,Z 603.479,A 0.000,B 0.000,C 90.000,E1 266.159} C_DIS
LIN {X 0.049,Y -410.822,Z 603.478,A 0.000,B 0.000,C 90.000,E1 266.102} C_DIS
LIN {X -0.010,Y -180.924,Z 603.478,A 0.000,B 0.000,C 90.000,E1 266.102} C_DIS
LIN {X -0.015,Y -180.899,Z 603.474,A 0.000,B 0.000,C 90.000,E1 265.241} C_DIS
LIN {X -0.065,Y -180.216,Z 603.464,A 0.000,B 0.000,C 90.000,E1 263.571} C_DIS
LIN {X 0.065,Y -179.034,Z 603.445,A 0.000,B 0.000,C 90.000,E1 260.151} C_DIS
LIN {X -0.049,Y -178.692,Z 603.441,A 0.000,B 0.000,C 90.000,E1 259.342} C_DIS
LIN {X 0.062,Y -175.741,Z 603.412,A 0.000,B 0.000,C 90.000,E1 254.212} C_DIS
LIN {X 0.057,Y -171.925,Z 603.384,A 0.000,B 0.000,C 90.000,E1 249.082} C_DIS
LIN {X 0.031,Y -171.299,Z 603.379,A 0.000,B 0.000,C 90.000,E1 248.230} C_DIS
LIN {X 0.077,Y -167.562,Z 603.355,A 0.000,B 0.000,C 90.000,E1 243.896} C_DIS
LIN {X 0.090,Y -166.187,Z 603.345,A 0.000,B 0.000,C 90.000,E1 242.153} C_DIS
LIN {X 0.080,Y -162.956,Z 603.326,A 0.000,B 0.000,C 90.000,E1 238.663} C_DIS
LIN {X -0.096,Y -160.865,Z 603.311,A 0.000,B 0.000,C 90.000,E1 236.087} C_DIS
LIN {X 0.008,Y -157.639,Z 603.292,A 0.000,B 0.000,C 90.000,E1 232.512} C_DIS
LIN {X 0.041,Y -155.677,Z 603.277,A 0.000,B 0.000,C 90.000,E1 229.828} C_DIS
LIN {X -0.013,Y -151.943,Z 603.252,A 0.000,B 0.000,C 90.000,E1 225.364} C_DIS
LIN {X -0.003,Y -150.182,Z 603.237,A 0.000,B 0.000,C 90.000,E1 222.651} C_DIS
LIN {X 0.027,Y -146.955,Z 603.212,A 0.000,B 0.000,C 90.000,E1 218.096} C_DIS
LIN {X -0.070,Y -145.543,Z 603.196,A 0.000,B 0.000,C 90.000,E1 215.391} C_DIS
LIN {X -0.069,Y -142.938,Z 603.171,A 0.000,B 0.000,C 90.000,E1 210.797} C_DIS
LIN {X -0.011,Y -141.563,Z 603.150,A 0.000,B 0.000,C 90.000,E1 207.078} C_DIS
LIN {X 0.041,Y -139.410,Z 603.114,A 0.000,B 0.000,C 90.000,E1 200.556} C_DIS
LIN {X -0.037,Y -139.131,Z 603.104,A 0.000,B 0.000,C 90.000,E1 198.725} C_DIS
LIN {X -0.010,Y -138.350,Z 603.057,A 0.000,B 0.000,C 90.000,E1 190.310} C_DIS
LIN {X -0.023,Y -139.497,Z 603.005,A 0.000,B 0.000,C 90.000,E1 180.974} C_DIS
LIN {X 0.058,Y -141.118,Z 602.974,A 0.000,B 0.000,C 90.000,E1 175.355} C_DIS
LIN {X 0.012,Y -142.497,Z 602.959,A 0.000,B 0.000,C 90.000,E1 172.591} C_DIS
LIN {X -0.042,Y -144.752,Z 602.933,A 0.000,B 0.000,C 90.000,E1 167.993} C_DIS
LIN {X 0.050,Y -147.361,Z 602.913,A 0.000,B 0.000,C 90.000,E1 164.283} C_DIS
LIN {X -0.028,Y -150.688,Z 602.887,A 0.000,B 0.000,C 90.000,E1 159.752} C_DIS
LIN {X 0.055,Y -154.168,Z 602.867,A 0.000,B 0.000,C 90.000,E1 156.102} C_DIS
LIN {X -0.015,Y -157.601,Z 602.847,A 0.000,B 0.000,C 90.000,E1 152.538} C_DIS
LIN {X -0.065,Y -161.853,Z 602.828,A 0.000,B 0.000,C 90.000,E1 148.997} C_DIS
LIN {X -0.047,Y -166.043,Z 602.808,A 0.000,B 0.000,C 90.000,E1 145.468} C_DIS
LIN {X -0.056,Y -171.047,Z 602.789,A 0.000,B 0.000,C 90.000,E1 141.984} C_DIS
LIN {X -0.025,Y -175.919,Z 602.770,A 0.000,B 0.000,C 90.000,E1 138.528} C_DIS
LIN {X -0.033,Y -180.156,Z 602.755,A 0.000,B 0.000,C 90.000,E1 135.972} C_DIS
LIN {X -0.064,Y -185.574,Z 602.737,A 0.000,B 0.000,C 90.000,E1 132.609} C_DIS
LIN {X -0.082,Y -191.285,Z 602.719,A 0.000,B 0.000,C 90.000,E1 129.483} C_DIS
LIN {X 0.063,Y -288.554,Z 602.719,A 0.000,B 0.000,C 90.000,E1 129.439} C_DIS
LIN {X -0.042,Y -289.936,Z 602.719,A 0.000,B 0.000,C 90.000,E1 129.439} C_DIS
LIN {X -0.094,Y -293.997,Z 602.718,A 0.000,B 0.000,C 90.000,E1 129.277} C_DIS
LIN {X 0.020,Y -297.211,Z 602.717,A 0.000,B 0.000,C 90.000,E1 128.991} C_DIS
LIN {X -0.170,Y -300.897,Z 602.714,A 0.000,B 0.000,C 90.000,E1 128.543} C_DIS
LIN {X 0.010,Y -302.668,Z 602.712,A 0.000,B 0.000,C 90.000,E1 128.177} C_DIS
LIN {X -0.047,Y -304.055,Z 602.710,A 0.000,B 0.000,C 90.000,E1 127.855} C_DIS
LIN {X 0.146,Y -307.867,Z 602.703,A 0.000,B 0.000,C 90.000,E1 126.503} C_DIS
LIN {X -0.062,Y -317.898,Z 602.685,A 0.000,B 0.000,C 90.000,E1 123.293} C_DIS
LIN {X -0.010,Y -328.242,Z 602.669,A 0.000,B 0.000,C 90.000,E1 120.413} C_DIS
LIN {X 0.015,Y -339.941,Z 602.653,A 0.000,B 0.000,C 90.000,E1 117.590} C_DIS
LIN {X 0.057,Y -353.092,Z 602.638,A 0.000,B 0.000,C 90.000,E1 114.823} C_DIS
LIN {X -0.203,Y -366.101,Z 602.625,A 0.000,B 0.000,C 90.000,E1 112.461} C_DIS
LIN {X 0.077,Y -380.450,Z 602.612,A 0.000,B 0.000,C 90.000,E1 110.066} C_DIS
LIN {X 0.113,Y -396.240,Z 602.599,A 0.000,B 0.000,C 90.000,E1 107.764} C_DIS
LIN {X -0.085,Y -413.588,Z 602.586,A 0.000,B 0.000,C 90.000,E1 105.552} C_DIS
LIN {X 0.036,Y -432.608,Z 602.574,A 0.000,B 0.000,C 90.000,E1 103.355} C_DIS
LIN {X 0.103,Y -452.718,Z 602.563,A 0.000,B 0.000,C 90.000,E1 101.299} C_DIS
LIN {X -0.083,Y -473.258,Z 602.552,A 0.000,B 0.000,C 90.000,E1 99.443} C_DIS
LIN {X 0.005,Y -475.168,Z 602.551,A 0.000,B 0.000,C 90.000,E1 99.208} C_DIS
LIN {X -0.133,Y -476.793,Z 602.550,A 0.000,B 0.000,C 90.000,E1 98.973} C_DIS
LIN {X 0.126,Y -478.012,Z 602.548,A 0.000,B 0.000,C 90.000,E1 98.690} C_DIS
LIN {X -0.136,Y -479.503,Z 602.546,A 0.000,B 0.000,C 90.000,E1 98.219} C_DIS
LIN {X 0.012,Y -479.952,Z 602.543,A 0.000,B 0.000,C 90.000,E1 97.701} C_DIS
LIN {X 0.171,Y -479.432,Z 602.540,A 0.000,B 0.000,C 90.000,E1 97.182} C_DIS
LIN {X -0.142,Y -477.861,Z 602.537,A 0.000,B 0.000,C 90.000,E1 96.720} C_DIS
LIN {X 0.201,Y -476.598,Z 602.536,A 0.000,B 0.000,C 90.000,E1 96.429} C_DIS
LIN {X 0.157,Y -471.210,Z 602.532,A 0.000,B 0.000,C 90.000,E1 95.682} C_DIS
LIN {X 0.216,Y -458.657,Z 602.522,A 0.000,B 0.000,C 90.000,E1 93.898} C_DIS
LIN {X 0.180,Y -446.010,Z 602.510,A 0.000,B 0.000,C 90.000,E1 91.835} C_DIS
LIN {X -0.125,Y -434.467,Z 602.499,A 0.000,B 0.000,C 90.000,E1 89.771} C_DIS
LIN {X 0.193,Y -426.942,Z 602.491,A 0.000,B 0.000,C 90.000,E1 88.396} C_DIS
LIN {X 0.107,Y -417.485,Z 602.482,A 0.000,B 0.000,C 90.000,E1 86.788} C_DIS
LIN {X 0.147,Y -401.886,Z 602.467,A 0.000,B 0.000,C 90.000,E1 84.033} C_DIS
LIN {X -0.095,Y -386.985,Z 602.451,A 0.000,B 0.000,C 90.000,E1 81.254} C_DIS
LIN {X 0.101,Y -375.445,Z 602.439,A 0.000,B 0.000,C 90.000,E1 78.926} C_DIS
LIN {X 0.080,Y -364.270,Z 602.426,A 0.000,B 0.000,C 90.000,E1 76.589} C_DIS
LIN {X -0.047,Y -349.736,Z 602.407,A 0.000,B 0.000,C 90.000,E1 73.323} C_DIS
LIN {X -0.019,Y -335.355,Z 602.387,A 0.000,B 0.000,C 90.000,E1 69.645} C_DIS
LIN {X 0.140,Y -323.656,Z 602.368,A 0.000,B 0.000,C 90.000,E1 66.177} C_DIS
LIN {X 0.101,Y -313.891,Z 602.350,A 0.000,B 0.000,C 90.000,E1 62.999} C_DIS
LIN {X -0.159,Y -306.504,Z 602.336,A 0.000,B 0.000,C 90.000,E1 60.461} C_DIS
LIN {X -0.093,Y -297.562,Z 602.318,A 0.000,B 0.000,C 90.000,E1 57.168} C_DIS
LIN {X 0.028,Y -290.832,Z 602.303,A 0.000,B 0.000,C 90.000,E1 54.482} C_DIS
LIN {X 0.068,Y -284.303,Z 602.288,A 0.000,B 0.000,C 90.000,E1 51.778} C_DIS
LIN {X 0.011,Y -279.324,Z 602.276,A 0.000,B 0.000,C 90.000,E1 49.747} C_DIS
LIN {X -0.135,Y -275.772,Z 602.269,A 0.000,B 0.000,C 90.000,E1 48.405} C_DIS
LIN {X 0.041,Y -271.938,Z 602.261,A 0.000,B 0.000,C 90.000,E1 46.986} C_DIS
LIN {X -0.018,Y -267.834,Z 602.253,A 0.000,B 0.000,C 90.000,E1 45.607} C_DIS
LIN {X -0.082,Y -262.321,Z 602.244,A 0.000,B 0.000,C 90.000,E1 43.866} C_DIS
LIN {X 0.036,Y -253.228,Z 602.228,A 0.000,B 0.000,C 90.000,E1 40.987} C_DIS
LIN {X -0.013,Y -243.361,Z 602.210,A 0.000,B 0.000,C 90.000,E1 37.729} C_DIS
LIN {X 0.001,Y -235.333,Z 602.193,A 0.000,B 0.000,C 90.000,E1 34.771} C_DIS
LIN {X 0.034,Y -226.405,Z 602.172,A 0.000,B 0.000,C 90.000,E1 31.003} C_DIS
LIN {X -0.079,Y -220.043,Z 602.155,A 0.000,B 0.000,C 90.000,E1 27.975} C_DIS
LIN {X 0.033,Y -214.432,Z 602.138,A 0.000,B 0.000,C 90.000,E1 24.847} C_DIS
LIN {X 0.019,Y -209.620,Z 602.121,A 0.000,B 0.000,C 90.000,E1 21.716} C_DIS
LIN {X -0.020,Y -204.632,Z 602.099,A 0.000,B 0.000,C 90.000,E1 17.764} C_DIS
LIN {X -0.060,Y -200.812,Z 602.076,A 0.000,B 0.000,C 90.000,E1 13.772} C_DIS
LIN {X -0.024,Y -197.549,Z 602.049,A 0.000,B 0.000,C 90.000,E1 8.916} C_DIS
LIN {X 0.050,Y -198.445,Z 601.952,A 0.000,B 0.000,C 90.000,E1 351.376} C_DIS
LIN {X 0.016,Y -202.069,Z 601.925,A 0.000,B 0.000,C 90.000,E1 346.533} C_DIS
LIN {X -0.067,Y -205.980,Z 601.903,A 0.000,B 0.000,C 90.000,E1 342.543} C_DIS
LIN {X 0.032,Y -210.778,Z 601.881,A 0.000,B 0.000,C 90.000,E1 338.539} C_DIS
LIN {X 0.092,Y -216.270,Z 601.859,A 0.000,B 0.000,C 90.000,E1 334.588} C_DIS
LIN {X 0.031,Y -222.471,Z 601.837,A 0.000,B 0.000,C 90.000,E1 330.717} C_DIS
LIN {X -0.098,Y -229.350,Z 601.816,A 0.000,B 0.000,C 90.000,E1 326.914} C_DIS
LIN {X -0.092,Y -236.607,Z 601.795,A 0.000,B 0.000,C 90.000,E1 323.130} C_DIS
LIN {X 0.013,Y -244.396,Z 601.774,A 0.000,B 0.000,C 90.000,E1 319.380} C_DIS
LIN {X -0.052,Y -252.962,Z 601.754,A 0.000,B 0.000,C 90.000,E1 315.729} C_DIS
LIN {X -0.031,Y -262.705,Z 601.734,A 0.000,B 0.000,C 90.000,E1 312.123} C_DIS
LIN {X 0.063,Y -271.637,Z 601.718,A 0.000,B 0.000,C 90.000,E1 309.277} C_DIS
LIN {X 0.117,Y -284.316,Z 601.699,A 0.000,B 0.000,C 90.000,E1 305.804} C_DIS
LIN {X 0.010,Y -294.075,Z 601.686,A 0.000,B 0.000,C 90.000,E1 303.452} C_DIS
LIN {X 0.043,Y -309.524,Z 601.667,A 0.000,B 0.000,C 90.000,E1 300.129} C_DIS
LIN {X -0.083,Y -322.601,Z 601.653,A 0.000,B 0.000,C 90.000,E1 297.564} C_DIS
LIN {X 0.065,Y -339.990,Z 601.636,A 0.000,B 0.000,C 90.000,E1 294.387} C_DIS
LIN {X -0.035,Y -355.287,Z 601.622,A 0.000,B 0.000,C 90.000,E1 291.950} C_DIS
LIN {X -0.110,Y -369.721,Z 601.610,A 0.000,B 0.000,C 90.000,E1 289.866} C_DIS
LIN {X -0.147,Y -394.694,Z 601.593,A 0.000,B 0.000,C 90.000,E1 286.677} C_DIS
LIN {X 0.001,Y -406.367,Z 601.585,A 0.000,B 0.000,C 90.000,E1 285.245} C_DIS
LIN {X -0.044,Y -420.211,Z 601.576,A 0.000,B 0.000,C 90.000,E1 283.592} C_DIS
LIN {X 0.142,Y -429.226,Z 601.569,A 0.000,B 0.000,C 90.000,E1 282.479} C_DIS
LIN {X -0.209,Y -439.949,Z 601.562,A 0.000,B 0.000,C 90.000,E1 281.186} C_DIS
LIN {X 0.142,Y -448.156,Z 601.556,A 0.000,B 0.000,C 90.000,E1 280.084} C_DIS
LIN {X -0.033,Y -457.660,Z 601.549,A 0.000,B 0.000,C 90.000,E1 278.803} C_DIS
LIN {X 0.089,Y -464.700,Z 601.543,A 0.000,B 0.000,C 90.000,E1 277.757} C_DIS
LIN {X -0.235,Y -471.175,Z 601.537,A 0.000,B 0.000,C 90.000,E1 276.777} C_DIS
LIN {X 0.185,Y -475.507,Z 601.533,A 0.000,B 0.000,C 90.000,E1 275.967} C_DIS
LIN {X 0.119,Y -479.175,Z 601.529,A 0.000,B 0.000,C 90.000,E1 275.220} C_DIS
LIN {X -0.211,Y -481.198,Z 601.526,A 0.000,B 0.000,C 90.000,E1 274.759} C_DIS
LIN {X -0.093,Y -482.878,Z 601.523,A 0.000,B 0.000,C 90.000,E1 274.245} C_DIS
LIN {X 0.073,Y -484.178,Z 601.521,A 0.000,B 0.000,C 90.000,E1 273.726} C_DIS
LIN {X 0.219,Y -485.147,Z 601.518,A 0.000,B 0.000,C 90.000,E1 273.212} C_DIS
LIN {X -0.084,Y -485.846,Z 601.515,A 0.000,B 0.000,C 90.000,E1 272.751} C_DIS
LIN {X 0.080,Y -486.201,Z 601.512,A 0.000,B 0.000,C 90.000,E1 272.236} C_DIS
LIN {X -0.222,Y -486.264,Z 601.510,A 0.000,B 0.000,C 90.000,E1 271.776} C_DIS
LIN {X -0.051,Y -485.953,Z 601.507,A 0.000,B 0.000,C 90.000,E1 271.260} C_DIS
LIN {X 0.120,Y -485.167,Z 601.504,A 0.000,B 0.000,C 90.000,E1 270.745} C_DIS
LIN {X -0.193,Y -483.848,Z 601.501,A 0.000,B 0.000,C 90.000,E1 270.286} C_DIS
LIN {X -0.027,Y -481.937,Z 601.499,A 0.000,B 0.000,C 90.000,E1 269.771} C_DIS
LIN {X 0.131,Y -479.242,Z 601.496,A 0.000,B 0.000,C 90.000,E1 269.255} C_DIS
LIN {X -0.040,Y -477.651,Z 601.495,A 0.000,B 0.000,C 90.000,E1 269.026} C_DIS
LIN {X 0.087,Y -473.678,Z 601.492,A 0.000,B 0.000,C 90.000,E1 268.511} C_DIS
LIN {X 0.208,Y -468.576,Z 601.489,A 0.000,B 0.000,C 90.000,E1 267.993} C_DIS
LIN {X 0.123,Y -462.482,Z 601.486,A 0.000,B 0.000,C 90.000,E1 267.535} C_DIS
LIN {X 0.223,Y -459.163,Z 601.485,A 0.000,B 0.000,C 90.000,E1 267.306} C_DIS
LIN {X 0.012,Y -452.012,Z 601.483,A 0.000,B 0.000,C 90.000,E1 266.963} C_DIS
LIN {X 0.002,Y -444.639,Z 601.482,A 0.000,B 0.000,C 90.000,E1 266.674} C_DIS
LIN {X 0.030,Y -437.067,Z 601.480,A 0.000,B 0.000,C 90.000,E1 266.445} C_DIS
LIN {X 0.029,Y -428.425,Z 601.479,A 0.000,B 0.000,C 90.000,E1 266.274} C_DIS
LIN {X 0.036,Y -418.861,Z 601.479,A 0.000,B 0.000,C 90.000,E1 266.159} C_DIS
LIN {X 0.017,Y -408.974,Z 601.478,A 0.000,B 0.000,C 90.000,E1 266.102} C_DIS
LIN {X -0.024,Y -180.924,Z 601.478,A 0.000,B 0.000,C 90.000,E1 266.102} C_DIS
LIN {X 0.020,Y -180.877,Z 601.473,A 0.000,B 0.000,C 90.000,E1 265.065} C_DIS
LIN {X -0.074,Y -178.943,Z 601.444,A 0.000,B 0.000,C 90.000,E1 259.859} C_DIS
LIN {X -0.030,Y -175.995,Z 601.415,A 0.000,B 0.000,C 90.000,E1 254.755} C_DIS
LIN {X -0.084,Y -175.499,Z 601.411,A 0.000,B 0.000,C 90.000,E1 253.921} C_DIS
LIN {X -0.022,Y -172.241,Z 601.387,A 0.000,B 0.000,C 90.000,E1 249.625} C_DIS
LIN {X -0.042,Y -171.719,Z 601.382,A 0.000,B 0.000,C 90.000,E1 248.773} C_DIS
LIN {X -0.033,Y -167.314,Z 601.353,A 0.000,B 0.000,C 90.000,E1 243.589} C_DIS
LIN {X 0.047,Y -166.696,Z 601.348,A 0.000,B 0.000,C 90.000,E1 242.692} C_DIS
LIN {X 0.038,Y -162.677,Z 601.324,A 0.000,B 0.000,C 90.000,E1 238.329} C_DIS
LIN {X 0.011,Y -161.367,Z 601.314,A 0.000,B 0.000,C 90.000,E1 236.580} C_DIS
LIN {X -0.080,Y -157.360,Z 601.290,A 0.000,B 0.000,C 90.000,E1 232.190} C_DIS
LIN {X 0.073,Y -155.350,Z 601.275,A 0.000,B 0.000,C 90.000,E1 229.461} C_DIS
LIN {X 0.003,Y -151.696,Z 601.250,A 0.000,B 0.000,C 90.000,E1 225.000} C_DIS
LIN {X 0.051,Y -150.557,Z 601.240,A 0.000,B 0.000,C 90.000,E1 223.176} C_DIS
LIN {X -0.033,Y -147.284,Z 601.215,A 0.000,B 0.000,C 90.000,E1 218.669} C_DIS
LIN {X -0.064,Y -145.313,Z 601.194,A 0.000,B 0.000,C 90.000,E1 215.025} C_DIS
LIN {X 0.046,Y -142.401,Z 601.164,A 0.000,B 0.000,C 90.000,E1 209.461} C_DIS
LIN {X 0.029,Y -141.384,Z 601.148,A 0.000,B 0.000,C 90.000,E1 206.693} C_DIS
LIN {X 0.021,Y -139.350,Z 601.112,A 0.000,B 0.000,C 90.000,E1 200.194} C_DIS
LIN {X 0.011,Y -138.788,Z 601.097,A 0.000,B 0.000,C 90.000,E1 197.402} C_DIS
LIN {X -0.067,Y -138.345,Z 601.055,A 0.000,B 0.000,C 90.000,E1 189.962} C_DIS
LIN {X -0.049,Y -139.384,Z 601.008,A 0.000,B 0.000,C 90.000,E1 181.547} C_DIS
LIN {X 0.004,Y -141.281,Z 600.972,A 0.000,B 0.000,C 90.000,E1 175.008} C_DIS
LIN {X -0.038,Y -142.645,Z 600.957,A 0.000,B 0.000,C 90.000,E1 172.243} C_DIS
LIN {X 0.054,Y -144.979,Z 600.931,A 0.000,B 0.000,C 90.000,E1 167.589} C_DIS
LIN {X 0.045,Y -147.606,Z 600.911,A 0.000,B 0.000,C 90.000,E1 163.921} C_DIS
LIN {X -0.018,Y -150.227,Z 600.891,A 0.000,B 0.000,C 90.000,E1 160.296} C_DIS
LIN {X -0.002,Y -153.618,Z 600.870,A 0.000,B 0.000,C 90.000,E1 156.666} C_DIS
LIN {X -0.015,Y -157.033,Z 600.850,A 0.000,B 0.000,C 90.000,E1 153.076} C_DIS
LIN {X -0.083,Y -161.158,Z 600.831,A 0.000,B 0.000,C 90.000,E1 149.537} C_DIS
LIN {X -0.001,Y -163.255,Z 600.821,A 0.000,B 0.000,C 90.000,E1 147.740} C_DIS
LIN {X 0.098,Y -167.692,Z 600.801,A 0.000,B 0.000,C 90.000,E1 144.196} C_DIS
LIN {X 0.012,Y -171.514,Z 600.787,A 0.000,B 0.000,C 90.000,E1 141.618} C_DIS
LIN {X 0.055,Y -176.449,Z 600.768,A 0.000,B 0.000,C 90.000,E1 138.162} C_DIS
LIN {X -0.075,Y -180.746,Z 600.753,A 0.000,B 0.000,C 90.000,E1 135.648} C_DIS
LIN {X 0.043,Y -186.151,Z 600.735,A 0.000,B 0.000,C 90.000,E1 132.243} C_DIS
LIN {X 0.041,Y -191.297,Z 600.719,A 0.000,B 0.000,C 90.000,E1 129.439} C_DIS
LIN {X 0.013,Y -288.548,Z 600.719,A 0.000,B 0.000,C 90.000,E1 129.439} C_DIS
LIN {X 0.054,Y -290.261,Z 600.719,A 0.000,B 0.000,C 90.000,E1 129.402} C_DIS
LIN {X -0.129,Y -295.115,Z 600.718,A 0.000,B 0.000,C 90.000,E1 129.197} C_DIS
LIN {X 0.103,Y -297.733,Z 600.716,A 0.000,B 0.000,C 90.000,E1 128.910} C_DIS
LIN {X 0.083,Y -301.501,Z 600.713,A 0.000,B 0.000,C 90.000,E1 128.382} C_DIS
LIN {X -0.159,Y -303.138,Z 600.711,A 0.000,B 0.000,C 90.000,E1 128.096} C_DIS
LIN {X 0.024,Y -304.425,Z 600.710,A 0.000,B 0.000,C 90.000,E1 127.729} C_DIS
LIN {X 0.113,Y -315.064,Z 600.690,A 0.000,B 0.000,C 90.000,E1 124.119} C_DIS
LIN {X -0.025,Y -325.029,Z 600.674,A 0.000,B 0.000,C 90.000,E1 121.258} C_DIS
LIN {X -0.096,Y -336.315,Z 600.658,A 0.000,B 0.000,C 90.000,E1 118.437} C_DIS
LIN {X -0.010,Y -349.027,Z 600.642,A 0.000,B 0.000,C 90.000,E1 115.643} C_DIS
LIN {X 0.100,Y -361.613,Z 600.629,A 0.000,B 0.000,C 90.000,E1 113.206} C_DIS
LIN {X -0.077,Y -375.506,Z 600.616,A 0.000,B 0.000,C 90.000,E1 110.865} C_DIS
LIN {X -0.044,Y -390.805,Z 600.603,A 0.000,B 0.000,C 90.000,E1 108.544} C_DIS
LIN {X 0.123,Y -407.622,Z 600.590,A 0.000,B 0.000,C 90.000,E1 106.260} C_DIS
LIN {X 0.089,Y -426.081,Z 600.578,A 0.000,B 0.000,C 90.000,E1 104.064} C_DIS
LIN {X 0.158,Y -445.959,Z 600.567,A 0.000,B 0.000,C 90.000,E1 101.951} C_DIS
LIN {X 0.164,Y -466.445,Z 600.556,A 0.000,B 0.000,C 90.000,E1 100.018} C_DIS
LIN {X 0.197,Y -471.647,Z 600.553,A 0.000,B 0.000,C 90.000,E1 99.557} C_DIS
LIN {X -0.176,Y -473.977,Z 600.552,A 0.000,B 0.000,C 90.000,E1 99.378} C_DIS
LIN {X -0.158,Y -475.739,Z 600.551,A 0.000,B 0.000,C 90.000,E1 99.151} C_DIS
LIN {X 0.175,Y -477.250,Z 600.549,A 0.000,B 0.000,C 90.000,E1 98.859} C_DIS
LIN {X 0.038,Y -478.380,Z 600.548,A 0.000,B 0.000,C 90.000,E1 98.624} C_DIS
LIN {X 0.180,Y -479.729,Z 600.545,A 0.000,B 0.000,C 90.000,E1 98.106} C_DIS
LIN {X -0.143,Y -480.055,Z 600.542,A 0.000,B 0.000,C 90.000,E1 97.644} C_DIS
LIN {X 0.019,Y -479.410,Z 600.540,A 0.000,B 0.000,C 90.000,E1 97.125} C_DIS
LIN {X 0.182,Y -477.693,Z 600.537,A 0.000,B 0.000,C 90.000,E1 96.606} C_DIS
LIN {X 0.050,Y -476.334,Z 600.535,A 0.000,B 0.000,C 90.000,E1 96.372} C_DIS
LIN {X 0.063,Y -458.290,Z 600.521,A 0.000,B 0.000,C 90.000,E1 93.841} C_DIS
LIN {X 0.039,Y -445.672,Z 600.510,A 0.000,B 0.000,C 90.000,E1 91.776} C_DIS
LIN {X -0.010,Y -435.586,Z 600.500,A 0.000,B 0.000,C 90.000,E1 89.943} C_DIS
LIN {X -0.109,Y -428.130,Z 600.492,A 0.000,B 0.000,C 90.000,E1 88.625} C_DIS
LIN {X -0.188,Y -418.687,Z 600.483,A 0.000,B 0.000,C 90.000,E1 87.020} C_DIS
LIN {X -0.128,Y -404.557,Z 600.470,A 0.000,B 0.000,C 90.000,E1 84.546} C_DIS
LIN {X 0.007,Y -389.557,Z 600.454,A 0.000,B 0.000,C 90.000,E1 81.724} C_DIS
LIN {X -0.101,Y -376.515,Z 600.440,A 0.000,B 0.000,C 90.000,E1 79.162} C_DIS
LIN {X -0.025,Y -363.907,Z 600.425,A 0.000,B 0.000,C 90.000,E1 76.520} C_DIS
LIN {X 0.188,Y -349.373,Z 600.407,A 0.000,B 0.000,C 90.000,E1 73.196} C_DIS
LIN {X -0.114,Y -335.052,Z 600.386,A 0.000,B 0.000,C 90.000,E1 69.571} C_DIS
LIN {X 0.051,Y -323.442,Z 600.367,A 0.000,B 0.000,C 90.000,E1 66.102} C_DIS
LIN {X 0.017,Y -313.707,Z 600.350,A 0.000,B 0.000,C 90.000,E1 62.922} C_DIS
LIN {X 0.026,Y -306.336,Z 600.335,A 0.000,B 0.000,C 90.000,E1 60.333} C_DIS
LIN {X 0.078,Y -297.395,Z 600.317,A 0.000,B 0.000,C 90.000,E1 57.041} C_DIS
LIN {X -0.050,Y -290.665,Z 600.302,A 0.000,B 0.000,C 90.000,E1 54.402} C_DIS
LIN {X -0.009,Y -284.138,Z 600.287,A 0.000,B 0.000,C 90.000,E1 51.698} C_DIS
LIN {X -0.066,Y -279.113,Z 600.276,A 0.000,B 0.000,C 90.000,E1 49.666} C_DIS
LIN {X 0.175,Y -275.564,Z 600.268,A 0.000,B 0.000,C 90.000,E1 48.243} C_DIS
LIN {X -0.038,Y -271.688,Z 600.261,A 0.000,B 0.000,C 90.000,E1 46.905} C_DIS
LIN {X 0.087,Y -267.546,Z 600.253,A 0.000,B 0.000,C 90.000,E1 45.486} C_DIS
LIN {X 0.068,Y -260.865,Z 600.241,A 0.000,B 0.000,C 90.000,E1 43.380} C_DIS
LIN {X -0.024,Y -251.753,Z 600.225,A 0.000,B 0.000,C 90.000,E1 40.539} C_DIS
LIN {X 0.079,Y -240.944,Z 600.205,A 0.000,B 0.000,C 90.000,E1 36.870} C_DIS
LIN {X 0.031,Y -233.206,Z 600.188,A 0.000,B 0.000,C 90.000,E1 33.913} C_DIS
LIN {X 0.059,Y -224.491,Z 600.167,A 0.000,B 0.000,C 90.000,E1 30.129} C_DIS
LIN {X -0.014,Y -218.347,Z 600.150,A 0.000,B 0.000,C 90.000,E1 27.078} C_DIS
LIN {X 0.053,Y -212.965,Z 600.133,A 0.000,B 0.000,C 90.000,E1 23.951} C_DIS
LIN {X 0.110,Y -208.388,Z 600.116,A 0.000,B 0.000,C 90.000,E1 20.791} C_DIS
LIN {X -0.037,Y -203.642,Z 600.094,A 0.000,B 0.000,C 90.000,E1 16.858} C_DIS
LIN {X 0.080,Y -199.458,Z 600.067,A 0.000,B 0.000,C 90.000,E1 12.007} C_DIS
LIN {X -0.047,Y -196.508,Z 600.035,A 0.000,B 0.000,C 90.000,E1 6.372} C_DIS
LIN {X 0.066,Y -197.583,Z 599.961,A 0.000,B 0.000,C 90.000,E1 352.996} C_DIS
LIN {X -0.076,Y -200.751,Z 599.934,A 0.000,B 0.000,C 90.000,E1 348.173} C_DIS
LIN {X 0.011,Y -205.140,Z 599.907,A 0.000,B 0.000,C 90.000,E1 343.323} C_DIS
LIN {X 0.016,Y -209.763,Z 599.885,A 0.000,B 0.000,C 90.000,E1 339.337} C_DIS
LIN {X -0.043,Y -215.140,Z 599.863,A 0.000,B 0.000,C 90.000,E1 335.409} C_DIS
LIN {X -0.049,Y -221.198,Z 599.842,A 0.000,B 0.000,C 90.000,E1 331.513} C_DIS
LIN {X -0.029,Y -227.944,Z 599.820,A 0.000,B 0.000,C 90.000,E1 327.661} C_DIS
LIN {X 0.026,Y -233.660,Z 599.803,A 0.000,B 0.000,C 90.000,E1 324.609} C_DIS
LIN {X -0.068,Y -241.165,Z 599.783,A 0.000,B 0.000,C 90.000,E1 320.884} C_DIS
LIN {X 0.130,Y -249.403,Z 599.762,A 0.000,B 0.000,C 90.000,E1 317.148} C_DIS
LIN {X 0.035,Y -258.600,Z 599.742,A 0.000,B 0.000,C 90.000,E1 313.542} C_DIS
LIN {X 0.056,Y -268.093,Z 599.724,A 0.000,B 0.000,C 90.000,E1 310.334} C_DIS
LIN {X -0.161,Y -279.020,Z 599.707,A 0.000,B 0.000,C 90.000,E1 307.237} C_DIS
LIN {X 0.045,Y -291.109,Z 599.690,A 0.000,B 0.000,C 90.000,E1 304.119} C_DIS
LIN {X -0.023,Y -306.224,Z 599.671,A 0.000,B 0.000,C 90.000,E1 300.797} C_DIS
LIN {X 0.052,Y -319.193,Z 599.657,A 0.000,B 0.000,C 90.000,E1 298.180} C_DIS
LIN {X -0.045,Y -336.275,Z 599.639,A 0.000,B 0.000,C 90.000,E1 295.027} C_DIS
LIN {X -0.079,Y -353.200,Z 599.624,A 0.000,B 0.000,C 90.000,E1 292.259} C_DIS
LIN {X -0.123,Y -369.676,Z 599.610,A 0.000,B 0.000,C 90.000,E1 289.866} C_DIS
LIN {X 0.172,Y -392.325,Z 599.594,A 0.000,B 0.000,C 90.000,E1 286.913} C_DIS
LIN {X -0.091,Y -404.020,Z 599.586,A 0.000,B 0.000,C 90.000,E1 285.536} C_DIS
LIN {X -0.185,Y -417.903,Z 599.577,A 0.000,B 0.000,C 90.000,E1 283.883} C_DIS
LIN {X 0.126,Y -429.286,Z 599.569,A 0.000,B 0.000,C 90.000,E1 282.479} C_DIS
LIN {X 0.207,Y -440.016,Z 599.562,A 0.000,B 0.000,C 90.000,E1 281.130} C_DIS
LIN {X 0.205,Y -448.214,Z 599.556,A 0.000,B 0.000,C 90.000,E1 280.074} C_DIS
LIN {X 0.217,Y -455.862,Z 599.550,A 0.000,B 0.000,C 90.000,E1 279.029} C_DIS
LIN {X -0.206,Y -463.011,Z 599.545,A 0.000,B 0.000,C 90.000,E1 278.049} C_DIS
LIN {X -0.027,Y -469.606,Z 599.539,A 0.000,B 0.000,C 90.000,E1 277.004} C_DIS
LIN {X -0.150,Y -474.095,Z 599.535,A 0.000,B 0.000,C 90.000,E1 276.258} C_DIS
LIN {X -0.224,Y -477.999,Z 599.530,A 0.000,B 0.000,C 90.000,E1 275.511} C_DIS
LIN {X 0.253,Y -481.169,Z 599.526,A 0.000,B 0.000,C 90.000,E1 274.702} C_DIS
LIN {X -0.109,Y -482.814,Z 599.523,A 0.000,B 0.000,C 90.000,E1 274.245} C_DIS
LIN {X 0.058,Y -484.152,Z 599.521,A 0.000,B 0.000,C 90.000,E1 273.726} C_DIS
LIN {X 0.204,Y -485.136,Z 599.518,A 0.000,B 0.000,C 90.000,E1 273.212} C_DIS
LIN {X -0.099,Y -485.851,Z 599.515,A 0.000,B 0.000,C 90.000,E1 272.751} C_DIS
LIN {X 0.063,Y -486.263,Z 599.512,A 0.000,B 0.000,C 90.000,E1 272.236} C_DIS
LIN {X 0.248,Y -486.298,Z 599.510,A 0.000,B 0.000,C 90.000,E1 271.718} C_DIS
LIN {X -0.068,Y -486.006,Z 599.507,A 0.000,B 0.000,C 90.000,E1 271.260} C_DIS
LIN {X 0.105,Y -485.227,Z 599.504,A 0.000,B 0.000,C 90.000,E1 270.745} C_DIS
LIN {X -0.208,Y -483.903,Z 599.501,A 0.000,B 0.000,C 90.000,E1 270.286} C_DIS
LIN {X -0.042,Y -481.963,Z 599.499,A 0.000,B 0.000,C 90.000,E1 269.771} C_DIS
LIN {X 0.116,Y -479.284,Z 599.496,A 0.000,B 0.000,C 90.000,E1 269.255} C_DIS
LIN {X -0.223,Y -475.800,Z 599.493,A 0.000,B 0.000,C 90.000,E1 268.797} C_DIS
LIN {X -0.104,Y -471.258,Z 599.490,A 0.000,B 0.000,C 90.000,E1 268.282} C_DIS
LIN {X 0.193,Y -468.538,Z 599.489,A 0.000,B 0.000,C 90.000,E1 267.993} C_DIS
LIN {X 0.107,Y -462.448,Z 599.486,A 0.000,B 0.000,C 90.000,E1 267.535} C_DIS
LIN {X 0.205,Y -459.083,Z 599.485,A 0.000,B 0.000,C 90.000,E1 267.306} C_DIS
LIN {X 0.114,Y -455.826,Z 599.484,A 0.000,B 0.000,C 90.000,E1 267.135} C_DIS
LIN {X -0.188,Y -448.632,Z 599.482,A 0.000,B 0.000,C 90.000,E1 266.846} C_DIS
LIN {X 0.021,Y -441.117,Z 599.481,A 0.000,B 0.000,C 90.000,E1 266.560} C_DIS
LIN {X -0.206,Y -433.242,Z 599.480,A 0.000,B 0.000,C 90.000,E1 266.388} C_DIS
LIN {X 0.003,Y -423.888,Z 599.479,A 0.000,B 0.000,C 90.000,E1 266.216} C_DIS
LIN {X 0.123,Y -412.584,Z 599.478,A 0.000,B 0.000,C 90.000,E1 266.102} C_DIS
LIN {X -0.020,Y -407.271,Z 599.478,A 0.000,B 0.000,C 90.000,E1 266.102} C_DIS
LIN {X -0.041,Y -180.924,Z 599.478,A 0.000,B 0.000,C 90.000,E1 266.102} C_DIS
LIN {X 0.004,Y -180.875,Z 599.473,A 0.000,B 0.000,C 90.000,E1 265.065} C_DIS
LIN {X 0.086,Y -178.941,Z 599.443,A 0.000,B 0.000,C 90.000,E1 259.803} C_DIS
LIN {X -0.047,Y -175.992,Z 599.415,A 0.000,B 0.000,C 90.000,E1 254.755} C_DIS
LIN {X 0.068,Y -175.495,Z 599.410,A 0.000,B 0.000,C 90.000,E1 253.866} C_DIS
LIN {X -0.038,Y -172.237,Z 599.387,A 0.000,B 0.000,C 90.000,E1 249.625} C_DIS
LIN {X -0.059,Y -171.715,Z 599.382,A 0.000,B 0.000,C 90.000,E1 248.773} C_DIS
LIN {X 0.026,Y -167.311,Z 599.353,A 0.000,B 0.000,C 90.000,E1 243.563} C_DIS
LIN {X 0.032,Y -166.691,Z 599.348,A 0.000,B 0.000,C 90.000,E1 242.692} C_DIS
LIN {X 0.022,Y -162.673,Z 599.324,A 0.000,B 0.000,C 90.000,E1 238.329} C_DIS
LIN {X -0.005,Y -161.362,Z 599.314,A 0.000,B 0.000,C 90.000,E1 236.580} C_DIS
LIN {X 0.029,Y -157.356,Z 599.290,A 0.000,B 0.000,C 90.000,E1 232.145} C_DIS
LIN {X 0.058,Y -155.345,Z 599.275,A 0.000,B 0.000,C 90.000,E1 229.461} C_DIS
LIN {X -0.013,Y -151.691,Z 599.250,A 0.000,B 0.000,C 90.000,E1 225.000} C_DIS
LIN {X 0.036,Y -150.554,Z 599.240,A 0.000,B 0.000,C 90.000,E1 223.176} C_DIS
LIN {X -0.048,Y -147.280,Z 599.215,A 0.000,B 0.000,C 90.000,E1 218.669} C_DIS
LIN {X 0.040,Y -145.309,Z 599.194,A 0.000,B 0.000,C 90.000,E1 214.978} C_DIS
LIN {X 0.031,Y -142.400,Z 599.164,A 0.000,B 0.000,C 90.000,E1 209.461} C_DIS
LIN {X 0.014,Y -141.381,Z 599.148,A 0.000,B 0.000,C 90.000,E1 206.693} C_DIS
LIN {X 0.055,Y -139.349,Z 599.112,A 0.000,B 0.000,C 90.000,E1 200.174} C_DIS
LIN {X -0.003,Y -138.786,Z 599.097,A 0.000,B 0.000,C 90.000,E1 197.402} C_DIS
LIN {X 0.055,Y -138.345,Z 599.055,A 0.000,B 0.000,C 90.000,E1 189.905} C_DIS
LIN {X -0.063,Y -139.387,Z 599.008,A 0.000,B 0.000,C 90.000,E1 181.547} C_DIS
LIN {X -0.011,Y -141.283,Z 598.972,A 0.000,B 0.000,C 90.000,E1 175.008} C_DIS
LIN {X -0.053,Y -142.647,Z 598.957,A 0.000,B 0.000,C 90.000,E1 172.243} C_DIS
LIN {X 0.039,Y -144.982,Z 598.931,A 0.000,B 0.000,C 90.000,E1 167.589} C_DIS
LIN {X 0.030,Y -147.610,Z 598.911,A 0.000,B 0.000,C 90.000,E1 163.921} C_DIS
LIN {X -0.032,Y -150.232,Z 598.890,A 0.000,B 0.000,C 90.000,E1 160.296} C_DIS
LIN {X -0.017,Y -153.624,Z 598.870,A 0.000,B 0.000,C 90.000,E1 156.666} C_DIS
LIN {X -0.030,Y -157.040,Z 598.850,A 0.000,B 0.000,C 90.000,E1 153.076} C_DIS
LIN {X 0.040,Y -161.164,Z 598.831,A 0.000,B 0.000,C 90.000,E1 149.488} C_DIS
LIN {X -0.017,Y -163.261,Z 598.821,A 0.000,B 0.000,C 90.000,E1 147.740} C_DIS
LIN {X 0.082,Y -167.700,Z 598.801,A 0.000,B 0.000,C 90.000,E1 144.196} C_DIS
LIN {X -0.005,Y -171.520,Z 598.787,A 0.000,B 0.000,C 90.000,E1 141.618} C_DIS
LIN {X 0.038,Y -176.458,Z 598.768,A 0.000,B 0.000,C 90.000,E1 138.162} C_DIS
LIN {X -0.091,Y -180.755,Z 598.753,A 0.000,B 0.000,C 90.000,E1 135.648} C_DIS
LIN {X 0.026,Y -186.160,Z 598.735,A 0.000,B 0.000,C 90.000,E1 132.243} C_DIS
LIN {X -0.009,Y -191.321,Z 598.719,A 0.000,B 0.000,C 90.000,E1 129.439} C_DIS
LIN {X -0.061,Y -289.061,Z 598.719,A 0.000,B 0.000,C 90.000,E1 129.439} C_DIS
LIN {X 0.027,Y -290.100,Z 598.719,A 0.000,B 0.000,C 90.000,E1 129.402} C_DIS
LIN {X -0.156,Y -295.066,Z 598.718,A 0.000,B 0.000,C 90.000,E1 129.197} C_DIS
LIN {X 0.077,Y -297.701,Z 598.716,A 0.000,B 0.000,C 90.000,E1 128.910} C_DIS
LIN {X 0.070,Y -301.467,Z 598.713,A 0.000,B 0.000,C 90.000,E1 128.382} C_DIS
LIN {X -0.172,Y -303.114,Z 598.711,A 0.000,B 0.000,C 90.000,E1 128.096} C_DIS
LIN {X 0.011,Y -304.407,Z 598.710,A 0.000,B 0.000,C 90.000,E1 127.729} C_DIS
LIN {X 0.099,Y -315.051,Z 598.690,A 0.000,B 0.000,C 90.000,E1 124.119} C_DIS
LIN {X -0.040,Y -325.017,Z 598.674,A 0.000,B 0.000,C 90.000,E1 121.258} C_DIS
LIN {X 0.048,Y -336.304,Z 598.658,A 0.000,B 0.000,C 90.000,E1 118.409} C_DIS
LIN {X -0.026,Y -349.017,Z 598.642,A 0.000,B 0.000,C 90.000,E1 115.643} C_DIS
LIN {X 0.083,Y -361.605,Z 598.629,A 0.000,B 0.000,C 90.000,E1 113.206} C_DIS
LIN {X 0.039,Y -375.499,Z 598.616,A 0.000,B 0.000,C 90.000,E1 110.844} C_DIS
LIN {X -0.063,Y -390.800,Z 598.603,A 0.000,B 0.000,C 90.000,E1 108.544} C_DIS
LIN {X 0.102,Y -407.618,Z 598.590,A 0.000,B 0.000,C 90.000,E1 106.260} C_DIS
LIN {X 0.067,Y -426.078,Z 598.578,A 0.000,B 0.000,C 90.000,E1 104.064} C_DIS
LIN {X 0.136,Y -445.959,Z 598.566,A 0.000,B 0.000,C 90.000,E1 101.951} C_DIS
LIN {X 0.142,Y -466.444,Z 598.556,A 0.000,B 0.000,C 90.000,E1 100.018} C_DIS
LIN {X 0.174,Y -471.647,Z 598.553,A 0.000,B 0.000,C 90.000,E1 99.557} C_DIS
LIN {X -0.198,Y -474.002,Z 598.552,A 0.000,B 0.000,C 90.000,E1 99.378} C_DIS
LIN {X -0.180,Y -475.788,Z 598.551,A 0.000,B 0.000,C 90.000,E1 99.151} C_DIS
LIN {X 0.154,Y -477.316,Z 598.549,A 0.000,B 0.000,C 90.000,E1 98.859} C_DIS
LIN {X 0.015,Y -478.461,Z 598.548,A 0.000,B 0.000,C 90.000,E1 98.624} C_DIS
LIN {X 0.159,Y -479.833,Z 598.545,A 0.000,B 0.000,C 90.000,E1 98.106} C_DIS
LIN {X -0.164,Y -480.179,Z 598.542,A 0.000,B 0.000,C 90.000,E1 97.644} C_DIS
LIN {X -0.002,Y -479.554,Z 598.540,A 0.000,B 0.000,C 90.000,E1 97.125} C_DIS
LIN {X 0.161,Y -477.860,Z 598.537,A 0.000,B 0.000,C 90.000,E1 96.606} C_DIS
LIN {X 0.031,Y -476.516,Z 598.535,A 0.000,B 0.000,C 90.000,E1 96.372} C_DIS
LIN {X -0.011,Y -461.880,Z 598.524,A 0.000,B 0.000,C 90.000,E1 94.359} C_DIS
LIN {X 0.078,Y -451.895,Z 598.516,A 0.000,B 0.000,C 90.000,E1 92.808} C_DIS
LIN {X -0.102,Y -439.978,Z 598.504,A 0.000,B 0.000,C 90.000,E1 90.745} C_DIS
LIN {X -0.130,Y -432.715,Z 598.497,A 0.000,B 0.000,C 90.000,E1 89.427} C_DIS
LIN {X 0.168,Y -425.089,Z 598.489,A 0.000,B 0.000,C 90.000,E1 88.051} C_DIS
LIN {X 0.133,Y -413.999,Z 598.479,A 0.000,B 0.000,C 90.000,E1 86.159} C_DIS
LIN {X 0.169,Y -397.030,Z 598.462,A 0.000,B 0.000,C 90.000,E1 83.109} C_DIS
LIN {X 0.152,Y -385.226,Z 598.449,A 0.000,B 0.000,C 90.000,E1 80.849} C_DIS
LIN {X -0.062,Y -372.300,Z 598.435,A 0.000,B 0.000,C 90.000,E1 78.285} C_DIS
LIN {X -0.054,Y -358.524,Z 598.419,A 0.000,B 0.000,C 90.000,E1 75.338} C_DIS
LIN {X 0.075,Y -344.444,Z 598.400,A 0.000,B 0.000,C 90.000,E1 72.000} C_DIS
LIN {X 0.161,Y -331.772,Z 598.381,A 0.000,B 0.000,C 90.000,E1 68.592} C_DIS
LIN {X -0.036,Y -321.504,Z 598.364,A 0.000,B 0.000,C 90.000,E1 65.485} C_DIS
LIN {X 0.006,Y -311.940,Z 598.346,A 0.000,B 0.000,C 90.000,E1 62.281} C_DIS
LIN {X 0.117,Y -304.595,Z 598.332,A 0.000,B 0.000,C 90.000,E1 59.665} C_DIS
LIN {X -0.134,Y -295.765,Z 598.313,A 0.000,B 0.000,C 90.000,E1 56.421} C_DIS
LIN {X 0.004,Y -287.448,Z 598.295,A 0.000,B 0.000,C 90.000,E1 53.050} C_DIS
LIN {X 0.051,Y -282.550,Z 598.283,A 0.000,B 0.000,C 90.000,E1 51.009} C_DIS
LIN {X -0.030,Y -277.400,Z 598.272,A 0.000,B 0.000,C 90.000,E1 48.976} C_DIS
LIN {X -0.014,Y -273.700,Z 598.264,A 0.000,B 0.000,C 90.000,E1 47.595} C_DIS
LIN {X -0.048,Y -269.684,Z 598.257,A 0.000,B 0.000,C 90.000,E1 46.215} C_DIS
LIN {X 0.110,Y -264.274,Z 598.247,A 0.000,B 0.000,C 90.000,E1 44.433} C_DIS
LIN {X -0.118,Y -256.283,Z 598.233,A 0.000,B 0.000,C 90.000,E1 42.000} C_DIS
LIN {X -0.125,Y -247.308,Z 598.217,A 0.000,B 0.000,C 90.000,E1 39.116} C_DIS
LIN {X -0.069,Y -238.915,Z 598.201,A 0.000,B 0.000,C 90.000,E1 36.171} C_DIS
LIN {X 0.032,Y -231.390,Z 598.184,A 0.000,B 0.000,C 90.000,E1 33.166} C_DIS
LIN {X 0.070,Y -224.492,Z 598.167,A 0.000,B 0.000,C 90.000,E1 30.129} C_DIS
LIN {X -0.003,Y -218.332,Z 598.150,A 0.000,B 0.000,C 90.000,E1 27.078} C_DIS
LIN {X 0.063,Y -212.949,Z 598.133,A 0.000,B 0.000,C 90.000,E1 23.951} C_DIS
LIN {X 0.119,Y -208.360,Z 598.116,A 0.000,B 0.000,C 90.000,E1 20.791} C_DIS
LIN {X -0.028,Y -203.629,Z 598.094,A 0.000,B 0.000,C 90.000,E1 16.858} C_DIS
LIN {X 0.089,Y -199.438,Z 598.067,A 0.000,B 0.000,C 90.000,E1 12.007} C_DIS
LIN {X -0.041,Y -196.488,Z 598.035,A 0.000,B 0.000,C 90.000,E1 6.372} C_DIS
LIN {X 0.067,Y -197.608,Z 597.961,A 0.000,B 0.000,C 90.000,E1 352.996} C_DIS
LIN {X -0.075,Y -200.778,Z 597.934,A 0.000,B 0.000,C 90.000,E1 348.173} C_DIS
LIN {X 0.013,Y -205.173,Z 597.907,A 0.000,B 0.000,C 90.000,E1 343.323} C_DIS
LIN {X 0.019,Y -209.777,Z 597.885,A 0.000,B 0.000,C 90.000,E1 339.337} C_DIS
LIN {X -0.039,Y -215.163,Z 597.863,A 0.000,B 0.000,C 90.000,E1 335.409} C_DIS
LIN {X -0.044,Y -221.214,Z 597.842,A 0.000,B 0.000,C 90.000,E1 331.513} C_DIS
LIN {X -0.023,Y -227.960,Z 597.820,A 0.000,B 0.000,C 90.000,E1 327.661} C_DIS
LIN {X 0.032,Y -233.650,Z 597.803,A 0.000,B 0.000,C 90.000,E1 324.609} C_DIS
LIN {X -0.062,Y -241.142,Z 597.783,A 0.000,B 0.000,C 90.000,E1 320.884} C_DIS
LIN {X 0.135,Y -249.369,Z 597.762,A 0.000,B 0.000,C 90.000,E1 317.148} C_DIS
LIN {X 0.040,Y -258.560,Z 597.742,A 0.000,B 0.000,C 90.000,E1 313.542} C_DIS
LIN {X 0.053,Y -268.037,Z 597.724,A 0.000,B 0.000,C 90.000,E1 310.334} C_DIS
LIN {X 0.003,Y -278.947,Z 597.707,A 0.000,B 0.000,C 90.000,E1 307.202} C_DIS
LIN {X 0.037,Y -291.059,Z 597.690,A 0.000,B 0.000,C 90.000,E1 304.119} C_DIS
LIN {X -0.033,Y -306.148,Z 597.671,A 0.000,B 0.000,C 90.000,E1 300.797} C_DIS
LIN {X 0.040,Y -319.111,Z 597.657,A 0.000,B 0.000,C 90.000,E1 298.180} C_DIS
LIN {X -0.061,Y -336.188,Z 597.639,A 0.000,B 0.000,C 90.000,E1 295.027} C_DIS
LIN {X 0.205,Y -351.134,Z 597.625,A 0.000,B 0.000,C 90.000,E1 292.514} C_DIS
LIN {X 0.128,Y -367.465,Z 597.612,A 0.000,B 0.000,C 90.000,E1 290.120} C_DIS
LIN {X 0.006,Y -389.962,Z 597.596,A 0.000,B 0.000,C 90.000,E1 287.221} C_DIS
LIN {X -0.116,Y -404.027,Z 597.586,A 0.000,B 0.000,C 90.000,E1 285.536} C_DIS
LIN {X -0.120,Y -417.828,Z 597.577,A 0.000,B 0.000,C 90.000,E1 283.883} C_DIS
LIN {X -0.227,Y -429.237,Z 597.569,A 0.000,B 0.000,C 90.000,E1 282.535} C_DIS
LIN {X 0.071,Y -437.896,Z 597.564,A 0.000,B 0.000,C 90.000,E1 281.422} C_DIS
LIN {X -0.246,Y -448.177,Z 597.556,A 0.000,B 0.000,C 90.000,E1 280.141} C_DIS
LIN {X -0.164,Y -455.854,Z 597.550,A 0.000,B 0.000,C 90.000,E1 279.086} C_DIS
LIN {X -0.137,Y -462.976,Z 597.545,A 0.000,B 0.000,C 90.000,E1 278.049} C_DIS
LIN {X 0.043,Y -469.534,Z 597.539,A 0.000,B 0.000,C 90.000,E1 277.004} C_DIS
LIN {X 0.241,Y -475.396,Z 597.533,A 0.000,B 0.000,C 90.000,E1 275.967} C_DIS
LIN {X 0.174,Y -479.065,Z 597.529,A 0.000,B 0.000,C 90.000,E1 275.220} C_DIS
LIN {X -0.155,Y -481.095,Z 597.526,A 0.000,B 0.000,C 90.000,E1 274.759} C_DIS
LIN {X -0.039,Y -482.739,Z 597.524,A 0.000,B 0.000,C 90.000,E1 274.245} C_DIS
LIN {X 0.128,Y -484.076,Z 597.521,A 0.000,B 0.000,C 90.000,E1 273.726} C_DIS
LIN {X -0.211,Y -485.110,Z 597.518,A 0.000,B 0.000,C 90.000,E1 273.269} C_DIS
LIN {X -0.030,Y -485.854,Z 597.515,A 0.000,B 0.000,C 90.000,E1 272.751} C_DIS
LIN {X 0.132,Y -486.266,Z 597.513,A 0.000,B 0.000,C 90.000,E1 272.236} C_DIS
LIN {X -0.169,Y -486.350,Z 597.510,A 0.000,B 0.000,C 90.000,E1 271.776} C_DIS
LIN {X 0.002,Y -486.060,Z 597.507,A 0.000,B 0.000,C 90.000,E1 271.260} C_DIS
LIN {X 0.174,Y -485.267,Z 597.504,A 0.000,B 0.000,C 90.000,E1 270.745} C_DIS
LIN {X -0.140,Y -483.948,Z 597.502,A 0.000,B 0.000,C 90.000,E1 270.286} C_DIS
LIN {X 0.028,Y -482.033,Z 597.499,A 0.000,B 0.000,C 90.000,E1 269.771} C_DIS
LIN {X 0.185,Y -479.369,Z 597.496,A 0.000,B 0.000,C 90.000,E1 269.255} C_DIS
LIN {X 0.016,Y -477.749,Z 597.495,A 0.000,B 0.000,C 90.000,E1 269.026} C_DIS
LIN {X 0.143,Y -473.748,Z 597.492,A 0.000,B 0.000,C 90.000,E1 268.511} C_DIS
LIN {X -0.197,Y -468.634,Z 597.489,A 0.000,B 0.000,C 90.000,E1 268.051} C_DIS
LIN {X 0.094,Y -465.586,Z 597.488,A 0.000,B 0.000,C 90.000,E1 267.764} C_DIS
LIN {X -0.198,Y -459.122,Z 597.485,A 0.000,B 0.000,C 90.000,E1 267.364} C_DIS
LIN {X 0.174,Y -455.948,Z 597.484,A 0.000,B 0.000,C 90.000,E1 267.135} C_DIS
LIN {X -0.137,Y -448.748,Z 597.482,A 0.000,B 0.000,C 90.000,E1 266.846} C_DIS
LIN {X 0.047,Y -441.258,Z 597.481,A 0.000,B 0.000,C 90.000,E1 266.560} C_DIS
LIN {X -0.196,Y -433.258,Z 597.480,A 0.000,B 0.000,C 90.000,E1 266.388} C_DIS
LIN {X 0.000,Y -423.970,Z 597.479,A 0.000,B 0.000,C 90.000,E1 266.216} C_DIS
LIN {X 0.119,Y -412.787,Z 597.478,A 0.000,B 0.000,C 90.000,E1 266.102} C_DIS
LIN {X -0.022,Y -407.435,Z 597.478,A 0.000,B 0.000,C 90.000,E1 266.102} C_DIS
LIN {X -0.041,Y -180.924,Z 597.478,A 0.000,B 0.000,C 90.000,E1 266.102} C_DIS
LIN {X 0.004,Y -180.875,Z 597.473,A 0.000,B 0.000,C 90.000,E1 265.065} C_DIS
LIN {X 0.087,Y -178.942,Z 597.443,A 0.000,B 0.000,C 90.000,E1 259.803} C_DIS
LIN {X -0.046,Y -175.992,Z 597.415,A 0.000,B 0.000,C 90.000,E1 254.755} C_DIS
LIN {X 0.069,Y -175.495,Z 597.410,A 0.000,B 0.000,C 90.000,E1 253.866} C_DIS
LIN {X -0.037,Y -172.238,Z 597.387,A 0.000,B 0.000,C 90.000,E1 249.625} C_DIS
LIN {X -0.059,Y -171.715,Z 597.382,A 0.000,B 0.000,C 90.000,E1 248.773} C_DIS
LIN {X 0.026,Y -167.311,Z 597.353,A 0.000,B 0.000,C 90.000,E1 243.563} C_DIS
LIN {X 0.032,Y -166.691,Z 597.348,A 0.000,B 0.000,C 90.000,E1 242.692} C_DIS
LIN {X 0.023,Y -162.672,Z 597.324,A 0.000,B 0.000,C 90.000,E1 238.329} C_DIS
LIN {X -0.004,Y -161.363,Z 597.314,A 0.000,B 0.000,C 90.000,E1 236.580} C_DIS
LIN {X 0.030,Y -157.356,Z 597.290,A 0.000,B 0.000,C 90.000,E1 232.145} C_DIS
LIN {X 0.058,Y -155.345,Z 597.275,A 0.000,B 0.000,C 90.000,E1 229.461} C_DIS
LIN {X -0.012,Y -151.692,Z 597.250,A 0.000,B 0.000,C 90.000,E1 225.000} C_DIS
LIN {X 0.036,Y -150.554,Z 597.240,A 0.000,B 0.000,C 90.000,E1 223.176} C_DIS
LIN {X -0.047,Y -147.281,Z 597.215,A 0.000,B 0.000,C 90.000,E1 218.669} C_DIS
LIN {X 0.040,Y -145.309,Z 597.194,A 0.000,B 0.000,C 90.000,E1 214.978} C_DIS
LIN {X 0.032,Y -142.399,Z 597.164,A 0.000,B 0.000,C 90.000,E1 209.461} C_DIS
LIN {X 0.015,Y -141.382,Z 597.148,A 0.000,B 0.000,C 90.000,E1 206.693} C_DIS
LIN {X 0.056,Y -139.349,Z 597.112,A 0.000,B 0.000,C 90.000,E1 200.174} C_DIS
LIN {X -0.002,Y -138.787,Z 597.097,A 0.000,B 0.000,C 90.000,E1 197.402} C_DIS
LIN {X 0.056,Y -138.344,Z 597.055,A 0.000,B 0.000,C 90.000,E1 189.905} C_DIS
LIN {X -0.063,Y -139.386,Z 597.008,A 0.000,B 0.000,C 90.000,E1 181.547} C_DIS
LIN {X -0.010,Y -141.283,Z 596.972,A 0.000,B 0.000,C 90.000,E1 175.008} C_DIS
LIN {X -0.052,Y -142.646,Z 596.957,A 0.000,B 0.000,C 90.000,E1 172.243} C_DIS
LIN {X 0.039,Y -144.982,Z 596.931,A 0.000,B 0.000,C 90.000,E1 167.589} C_DIS
LIN {X 0.030,Y -147.610,Z 596.911,A 0.000,B 0.000,C 90.000,E1 163.921} C_DIS
LIN {X -0.032,Y -150.232,Z 596.890,A 0.000,B 0.000,C 90.000,E1 160.296} C_DIS
LIN {X -0.017,Y -153.624,Z 596.870,A 0.000,B 0.000,C 90.000,E1 156.666} C_DIS
LIN {X -0.029,Y -157.040,Z 596.850,A 0.000,B 0.000,C 90.000,E1 153.076} C_DIS
LIN {X 0.040,Y -161.165,Z 596.831,A 0.000,B 0.000,C 90.000,E1 149.488} C_DIS
LIN {X -0.017,Y -163.260,Z 596.821,A 0.000,B 0.000,C 90.000,E1 147.740} C_DIS
LIN {X 0.082,Y -167.699,Z 596.801,A 0.000,B 0.000,C 90.000,E1 144.196} C_DIS
LIN {X -0.005,Y -171.520,Z 596.787,A 0.000,B 0.000,C 90.000,E1 141.618} C_DIS
LIN {X 0.038,Y -176.458,Z 596.768,A 0.000,B 0.000,C 90.000,E1 138.162} C_DIS
LIN {X -0.091,Y -180.754,Z 596.753,A 0.000,B 0.000,C 90.000,E1 135.648} C_DIS
LIN {X 0.027,Y -186.159,Z 596.735,A 0.000,B 0.000,C 90.000,E1 132.243} C_DIS
LIN {X -0.040,Y -191.337,Z 596.719,A 0.000,B 0.000,C 90.000,E1 129.439} C_DIS
LIN {X 0.075,Y -289.060,Z 596.719,A 0.000,B 0.000,C 90.000,E1 129.402} C_DIS
LIN {X -0.155,Y -294.943,Z 596.718,A 0.000,B 0.000,C 90.000,E1 129.197} C_DIS
LIN {X 0.078,Y -297.617,Z 596.716,A 0.000,B 0.000,C 90.000,E1 128.910} C_DIS
LIN {X 0.105,Y -301.381,Z 596.713,A 0.000,B 0.000,C 90.000,E1 128.382} C_DIS
LIN {X -0.137,Y -303.049,Z 596.711,A 0.000,B 0.000,C 90.000,E1 128.096} C_DIS
LIN {X 0.046,Y -304.357,Z 596.710,A 0.000,B 0.000,C 90.000,E1 127.729} C_DIS
LIN {X 0.134,Y -315.011,Z 596.690,A 0.000,B 0.000,C 90.000,E1 124.119} C_DIS
LIN {X -0.005,Y -324.973,Z 596.674,A 0.000,B 0.000,C 90.000,E1 121.258} C_DIS
LIN {X -0.077,Y -336.257,Z 596.658,A 0.000,B 0.000,C 90.000,E1 118.437} C_DIS
LIN {X -0.143,Y -348.967,Z 596.642,A 0.000,B 0.000,C 90.000,E1 115.668} C_DIS
LIN {X 0.117,Y -361.551,Z 596.629,A 0.000,B 0.000,C 90.000,E1 113.206} C_DIS
LIN {X -0.060,Y -375.442,Z 596.616,A 0.000,B 0.000,C 90.000,E1 110.865} C_DIS
LIN {X -0.029,Y -390.738,Z 596.603,A 0.000,B 0.000,C 90.000,E1 108.544} C_DIS
LIN {X 0.137,Y -407.553,Z 596.590,A 0.000,B 0.000,C 90.000,E1 106.260} C_DIS
LIN {X 0.102,Y -426.010,Z 596.578,A 0.000,B 0.000,C 90.000,E1 104.064} C_DIS
LIN {X 0.169,Y -445.888,Z 596.567,A 0.000,B 0.000,C 90.000,E1 101.951} C_DIS
LIN {X 0.173,Y -466.373,Z 596.556,A 0.000,B 0.000,C 90.000,E1 100.018} C_DIS
LIN {X -0.168,Y -473.971,Z 596.552,A 0.000,B 0.000,C 90.000,E1 99.378} C_DIS
LIN {X -0.152,Y -475.792,Z 596.551,A 0.000,B 0.000,C 90.000,E1 99.151} C_DIS
LIN {X 0.182,Y -477.349,Z 596.549,A 0.000,B 0.000,C 90.000,E1 98.859} C_DIS
LIN {X 0.044,Y -478.516,Z 596.548,A 0.000,B 0.000,C 90.000,E1 98.624} C_DIS
LIN {X 0.189,Y -479.924,Z 596.545,A 0.000,B 0.000,C 90.000,E1 98.106} C_DIS
LIN {X -0.135,Y -480.301,Z 596.542,A 0.000,B 0.000,C 90.000,E1 97.644} C_DIS
LIN {X 0.028,Y -479.708,Z 596.540,A 0.000,B 0.000,C 90.000,E1 97.125} C_DIS
LIN {X 0.192,Y -478.051,Z 596.537,A 0.000,B 0.000,C 90.000,E1 96.606} C_DIS
LIN {X 0.062,Y -476.732,Z 596.535,A 0.000,B 0.000,C 90.000,E1 96.372} C_DIS
LIN {X -0.129,Y -469.373,Z 596.530,A 0.000,B 0.000,C 90.000,E1 95.391} C_DIS
LIN {X -0.132,Y -456.913,Z 596.520,A 0.000,B 0.000,C 90.000,E1 93.612} C_DIS
LIN {X 0.067,Y -445.899,Z 596.510,A 0.000,B 0.000,C 90.000,E1 91.776} C_DIS
LIN {X 0.183,Y -434.331,Z 596.498,A 0.000,B 0.000,C 90.000,E1 89.656} C_DIS
LIN {X 0.210,Y -425.215,Z 596.489,A 0.000,B 0.000,C 90.000,E1 88.051} C_DIS
LIN {X 0.176,Y -414.094,Z 596.479,A 0.000,B 0.000,C 90.000,E1 86.159} C_DIS
LIN {X -0.180,Y -397.133,Z 596.462,A 0.000,B 0.000,C 90.000,E1 83.166} C_DIS
LIN {X 0.197,Y -385.324,Z 596.449,A 0.000,B 0.000,C 90.000,E1 80.849} C_DIS
LIN {X -0.026,Y -373.806,Z 596.437,A 0.000,B 0.000,C 90.000,E1 78.578} C_DIS
LIN {X -0.028,Y -361.261,Z 596.422,A 0.000,B 0.000,C 90.000,E1 75.936} C_DIS
LIN {X 0.105,Y -345.689,Z 596.402,A 0.000,B 0.000,C 90.000,E1 72.308} C_DIS
LIN {X -0.103,Y -331.820,Z 596.381,A 0.000,B 0.000,C 90.000,E1 68.646} C_DIS
LIN {X 0.010,Y -321.599,Z 596.364,A 0.000,B 0.000,C 90.000,E1 65.485} C_DIS
LIN {X 0.053,Y -312.043,Z 596.346,A 0.000,B 0.000,C 90.000,E1 62.281} C_DIS
LIN {X 0.167,Y -304.701,Z 596.332,A 0.000,B 0.000,C 90.000,E1 59.665} C_DIS
LIN {X -0.084,Y -295.865,Z 596.313,A 0.000,B 0.000,C 90.000,E1 56.421} C_DIS
LIN {X 0.056,Y -287.531,Z 596.295,A 0.000,B 0.000,C 90.000,E1 53.050} C_DIS
LIN {X 0.104,Y -282.617,Z 596.284,A 0.000,B 0.000,C 90.000,E1 51.009} C_DIS
LIN {X 0.023,Y -277.452,Z 596.272,A 0.000,B 0.000,C 90.000,E1 48.976} C_DIS
LIN {X 0.038,Y -273.740,Z 596.264,A 0.000,B 0.000,C 90.000,E1 47.595} C_DIS
LIN {X 0.005,Y -269.700,Z 596.257,A 0.000,B 0.000,C 90.000,E1 46.215} C_DIS
LIN {X 0.035,Y -263.174,Z 596.245,A 0.000,B 0.000,C 90.000,E1 44.109} C_DIS
LIN {X -0.031,Y -255.159,Z 596.231,A 0.000,B 0.000,C 90.000,E1 41.634} C_DIS
LIN {X -0.058,Y -245.155,Z 596.213,A 0.000,B 0.000,C 90.000,E1 38.382} C_DIS
LIN {X -0.054,Y -236.971,Z 596.197,A 0.000,B 0.000,C 90.000,E1 35.438} C_DIS
LIN {X 0.055,Y -229.598,Z 596.180,A 0.000,B 0.000,C 90.000,E1 32.418} C_DIS
LIN {X -0.062,Y -222.888,Z 596.163,A 0.000,B 0.000,C 90.000,E1 29.411} C_DIS
LIN {X 0.024,Y -216.920,Z 596.146,A 0.000,B 0.000,C 90.000,E1 26.309} C_DIS
LIN {X -0.035,Y -211.692,Z 596.129,A 0.000,B 0.000,C 90.000,E1 23.206} C_DIS
LIN {X -0.063,Y -206.325,Z 596.107,A 0.000,B 0.000,C 90.000,E1 19.268} C_DIS
LIN {X 0.057,Y -202.060,Z 596.085,A 0.000,B 0.000,C 90.000,E1 15.245} C_DIS
LIN {X -0.020,Y -198.332,Z 596.058,A 0.000,B 0.000,C 90.000,E1 10.433} C_DIS
LIN {X -0.086,Y -195.841,Z 596.022,A 0.000,B 0.000,C 90.000,E1 3.955} C_DIS
LIN {X 0.101,Y -197.241,Z 595.966,A 0.000,B 0.000,C 90.000,E1 353.799} C_DIS
LIN {X -0.076,Y -200.158,Z 595.939,A 0.000,B 0.000,C 90.000,E1 348.982} C_DIS
LIN {X -0.103,Y -204.382,Z 595.912,A 0.000,B 0.000,C 90.000,E1 344.157} C_DIS
LIN {X 0.009,Y -208.813,Z 595.890,A 0.000,B 0.000,C 90.000,E1 340.134} C_DIS
LIN {X 0.028,Y -214.032,Z 595.868,A 0.000,B 0.000,C 90.000,E1 336.177} C_DIS
LIN {X -0.013,Y -219.975,Z 595.846,A 0.000,B 0.000,C 90.000,E1 332.281} C_DIS
LIN {X 0.054,Y -226.577,Z 595.825,A 0.000,B 0.000,C 90.000,E1 328.408} C_DIS
LIN {X -0.056,Y -232.216,Z 595.808,A 0.000,B 0.000,C 90.000,E1 325.388} C_DIS
LIN {X -0.009,Y -239.583,Z 595.787,A 0.000,B 0.000,C 90.000,E1 321.618} C_DIS
LIN {X -0.025,Y -247.619,Z 595.766,A 0.000,B 0.000,C 90.000,E1 317.919} C_DIS
LIN {X 0.006,Y -256.589,Z 595.746,A 0.000,B 0.000,C 90.000,E1 314.271} C_DIS
LIN {X -0.069,Y -265.754,Z 595.728,A 0.000,B 0.000,C 90.000,E1 311.067} C_DIS
LIN {X -0.064,Y -275.099,Z 595.712,A 0.000,B 0.000,C 90.000,E1 308.257} C_DIS
LIN {X -0.072,Y -288.175,Z 595.693,A 0.000,B 0.000,C 90.000,E1 304.818} C_DIS
LIN {X -0.095,Y -301.437,Z 595.677,A 0.000,B 0.000,C 90.000,E1 301.799} C_DIS
LIN {X 0.117,Y -317.385,Z 595.658,A 0.000,B 0.000,C 90.000,E1 298.487} C_DIS
LIN {X -0.044,Y -334.314,Z 595.641,A 0.000,B 0.000,C 90.000,E1 295.335} C_DIS
LIN {X 0.169,Y -349.106,Z 595.627,A 0.000,B 0.000,C 90.000,E1 292.823} C_DIS
LIN {X 0.113,Y -367.405,Z 595.612,A 0.000,B 0.000,C 90.000,E1 290.120} C_DIS
LIN {X -0.011,Y -389.940,Z 595.596,A 0.000,B 0.000,C 90.000,E1 287.221} C_DIS
LIN {X 0.069,Y -401.702,Z 595.588,A 0.000,B 0.000,C 90.000,E1 285.788} C_DIS
LIN {X 0.050,Y -415.642,Z 595.578,A 0.000,B 0.000,C 90.000,E1 284.120} C_DIS
LIN {X -0.079,Y -427.175,Z 595.571,A 0.000,B 0.000,C 90.000,E1 282.771} C_DIS
LIN {X -0.231,Y -435.947,Z 595.565,A 0.000,B 0.000,C 90.000,E1 281.715} C_DIS
LIN {X -0.069,Y -446.341,Z 595.558,A 0.000,B 0.000,C 90.000,E1 280.366} C_DIS
LIN {X 0.172,Y -456.007,Z 595.550,A 0.000,B 0.000,C 90.000,E1 279.029} C_DIS
LIN {X 0.210,Y -463.071,Z 595.545,A 0.000,B 0.000,C 90.000,E1 277.992} C_DIS
LIN {X -0.071,Y -469.607,Z 595.539,A 0.000,B 0.000,C 90.000,E1 277.004} C_DIS
LIN {X -0.192,Y -474.057,Z 595.535,A 0.000,B 0.000,C 90.000,E1 276.258} C_DIS
LIN {X 0.208,Y -477.954,Z 595.530,A 0.000,B 0.000,C 90.000,E1 275.454} C_DIS
LIN {X 0.209,Y -481.147,Z 595.526,A 0.000,B 0.000,C 90.000,E1 274.702} C_DIS
LIN {X -0.154,Y -482.773,Z 595.523,A 0.000,B 0.000,C 90.000,E1 274.245} C_DIS
LIN {X 0.014,Y -484.109,Z 595.521,A 0.000,B 0.000,C 90.000,E1 273.726} C_DIS
LIN {X 0.159,Y -485.157,Z 595.518,A 0.000,B 0.000,C 90.000,E1 273.212} C_DIS
LIN {X -0.145,Y -485.898,Z 595.515,A 0.000,B 0.000,C 90.000,E1 272.751} C_DIS
LIN {X 0.019,Y -486.304,Z 595.512,A 0.000,B 0.000,C 90.000,E1 272.236} C_DIS
LIN {X 0.203,Y -486.416,Z 595.510,A 0.000,B 0.000,C 90.000,E1 271.718} C_DIS
LIN {X -0.112,Y -486.073,Z 595.507,A 0.000,B 0.000,C 90.000,E1 271.260} C_DIS
LIN {X 0.061,Y -485.260,Z 595.504,A 0.000,B 0.000,C 90.000,E1 270.745} C_DIS
LIN {X 0.232,Y -483.927,Z 595.501,A 0.000,B 0.000,C 90.000,E1 270.229} C_DIS
LIN {X -0.085,Y -481.995,Z 595.499,A 0.000,B 0.000,C 90.000,E1 269.771} C_DIS
LIN {X 0.073,Y -479.345,Z 595.496,A 0.000,B 0.000,C 90.000,E1 269.255} C_DIS
LIN {X 0.211,Y -475.777,Z 595.493,A 0.000,B 0.000,C 90.000,E1 268.740} C_DIS
LIN {X -0.145,Y -471.190,Z 595.490,A 0.000,B 0.000,C 90.000,E1 268.282} C_DIS
LIN {X 0.155,Y -468.465,Z 595.489,A 0.000,B 0.000,C 90.000,E1 267.993} C_DIS
LIN {X -0.029,Y -465.380,Z 595.488,A 0.000,B 0.000,C 90.000,E1 267.764} C_DIS
LIN {X 0.158,Y -458.959,Z 595.485,A 0.000,B 0.000,C 90.000,E1 267.306} C_DIS
LIN {X -0.028,Y -451.877,Z 595.483,A 0.000,B 0.000,C 90.000,E1 266.963} C_DIS
LIN {X -0.036,Y -444.416,Z 595.482,A 0.000,B 0.000,C 90.000,E1 266.674} C_DIS
LIN {X -0.014,Y -436.829,Z 595.480,A 0.000,B 0.000,C 90.000,E1 266.445} C_DIS
LIN {X -0.027,Y -428.034,Z 595.479,A 0.000,B 0.000,C 90.000,E1 266.274} C_DIS
LIN {X -0.026,Y -418.308,Z 595.479,A 0.000,B 0.000,C 90.000,E1 266.159} C_DIS
LIN {X -0.041,Y -407.030,Z 595.478,A 0.000,B 0.000,C 90.000,E1 266.102} C_DIS
LIN {X -0.049,Y -180.924,Z 595.478,A 0.000,B 0.000,C 90.000,E1 266.102} C_DIS
LIN {X -0.004,Y -180.875,Z 595.473,A 0.000,B 0.000,C 90.000,E1 265.065} C_DIS
LIN {X 0.078,Y -178.941,Z 595.443,A 0.000,B 0.000,C 90.000,E1 259.803} C_DIS
LIN {X -0.054,Y -175.991,Z 595.415,A 0.000,B 0.000,C 90.000,E1 254.755} C_DIS
LIN {X 0.061,Y -175.492,Z 595.410,A 0.000,B 0.000,C 90.000,E1 253.866} C_DIS
LIN {X -0.045,Y -172.236,Z 595.387,A 0.000,B 0.000,C 90.000,E1 249.625} C_DIS
LIN {X -0.067,Y -171.714,Z 595.382,A 0.000,B 0.000,C 90.000,E1 248.773} C_DIS
LIN {X 0.018,Y -167.309,Z 595.353,A 0.000,B 0.000,C 90.000,E1 243.563} C_DIS
LIN {X 0.024,Y -166.690,Z 595.348,A 0.000,B 0.000,C 90.000,E1 242.692} C_DIS
LIN {X 0.014,Y -162.670,Z 595.324,A 0.000,B 0.000,C 90.000,E1 238.329} C_DIS
LIN {X -0.012,Y -161.361,Z 595.314,A 0.000,B 0.000,C 90.000,E1 236.580} C_DIS
LIN {X 0.022,Y -157.354,Z 595.290,A 0.000,B 0.000,C 90.000,E1 232.145} C_DIS
LIN {X 0.051,Y -155.342,Z 595.275,A 0.000,B 0.000,C 90.000,E1 229.461} C_DIS
LIN {X -0.020,Y -151.690,Z 595.250,A 0.000,B 0.000,C 90.000,E1 225.000} C_DIS
LIN {X 0.028,Y -150.553,Z 595.240,A 0.000,B 0.000,C 90.000,E1 223.176} C_DIS
LIN {X -0.054,Y -147.279,Z 595.215,A 0.000,B 0.000,C 90.000,E1 218.669} C_DIS
LIN {X 0.033,Y -145.307,Z 595.194,A 0.000,B 0.000,C 90.000,E1 214.978} C_DIS
LIN {X 0.025,Y -142.398,Z 595.164,A 0.000,B 0.000,C 90.000,E1 209.461} C_DIS
LIN {X 0.007,Y -141.380,Z 595.148,A 0.000,B 0.000,C 90.000,E1 206.693} C_DIS
LIN {X 0.049,Y -139.349,Z 595.112,A 0.000,B 0.000,C 90.000,E1 200.174} C_DIS
LIN {X -0.009,Y -138.785,Z 595.097,A 0.000,B 0.000,C 90.000,E1 197.402} C_DIS
LIN {X 0.049,Y -138.344,Z 595.055,A 0.000,B 0.000,C 90.000,E1 189.905} C_DIS
LIN {X 0.069,Y -139.388,Z 595.008,A 0.000,B 0.000,C 90.000,E1 181.489} C_DIS
LIN {X -0.017,Y -141.284,Z 594.972,A 0.000,B 0.000,C 90.000,E1 175.008} C_DIS
LIN {X -0.059,Y -142.647,Z 594.957,A 0.000,B 0.000,C 90.000,E1 172.243} C_DIS
LIN {X 0.033,Y -144.984,Z 594.931,A 0.000,B 0.000,C 90.000,E1 167.589} C_DIS
LIN {X 0.022,Y -147.611,Z 594.911,A 0.000,B 0.000,C 90.000,E1 163.921} C_DIS
LIN {X -0.040,Y -150.234,Z 594.890,A 0.000,B 0.000,C 90.000,E1 160.296} C_DIS
LIN {X -0.025,Y -153.627,Z 594.870,A 0.000,B 0.000,C 90.000,E1 156.666} C_DIS
LIN {X -0.037,Y -157.042,Z 594.850,A 0.000,B 0.000,C 90.000,E1 153.076} C_DIS
LIN {X 0.033,Y -161.168,Z 594.831,A 0.000,B 0.000,C 90.000,E1 149.488} C_DIS
LIN {X -0.024,Y -163.264,Z 594.821,A 0.000,B 0.000,C 90.000,E1 147.740} C_DIS
LIN {X 0.074,Y -167.704,Z 594.801,A 0.000,B 0.000,C 90.000,E1 144.196} C_DIS
LIN {X -0.012,Y -171.524,Z 594.787,A 0.000,B 0.000,C 90.000,E1 141.618} C_DIS
LIN {X 0.030,Y -176.462,Z 594.768,A 0.000,B 0.000,C 90.000,E1 138.162} C_DIS
LIN {X -0.099,Y -180.758,Z 594.753,A 0.000,B 0.000,C 90.000,E1 135.648} C_DIS
LIN {X 0.018,Y -186.165,Z 594.735,A 0.000,B 0.000,C 90.000,E1 132.243} C_DIS
LIN {X -0.049,Y -191.341,Z 594.719,A 0.000,B 0.000,C 90.000,E1 129.439} C_DIS
LIN {X 0.061,Y -288.367,Z 594.719,A 0.000,B 0.000,C 90.000,E1 129.402} C_DIS
LIN {X 0.014,Y -289.256,Z 594.719,A 0.000,B 0.000,C 90.000,E1 129.402} C_DIS
LIN {X -0.169,Y -294.854,Z 594.718,A 0.000,B 0.000,C 90.000,E1 129.197} C_DIS
LIN {X 0.064,Y -297.558,Z 594.716,A 0.000,B 0.000,C 90.000,E1 128.910} C_DIS
LIN {X 0.116,Y -301.320,Z 594.713,A 0.000,B 0.000,C 90.000,E1 128.382} C_DIS
LIN {X -0.126,Y -303.003,Z 594.711,A 0.000,B 0.000,C 90.000,E1 128.096} C_DIS
LIN {X 0.057,Y -304.322,Z 594.710,A 0.000,B 0.000,C 90.000,E1 127.729} C_DIS
LIN {X 0.144,Y -314.984,Z 594.690,A 0.000,B 0.000,C 90.000,E1 124.119} C_DIS
LIN {X 0.004,Y -324.946,Z 594.674,A 0.000,B 0.000,C 90.000,E1 121.258} C_DIS
LIN {X -0.069,Y -336.228,Z 594.658,A 0.000,B 0.000,C 90.000,E1 118.437} C_DIS
LIN {X -0.135,Y -348.937,Z 594.642,A 0.000,B 0.000,C 90.000,E1 115.668} C_DIS
LIN {X 0.125,Y -361.521,Z 594.629,A 0.000,B 0.000,C 90.000,E1 113.206} C_DIS
LIN {X -0.053,Y -375.410,Z 594.616,A 0.000,B 0.000,C 90.000,E1 110.865} C_DIS
LIN {X -0.021,Y -390.706,Z 594.603,A 0.000,B 0.000,C 90.000,E1 108.544} C_DIS
LIN {X 0.143,Y -407.520,Z 594.590,A 0.000,B 0.000,C 90.000,E1 106.260} C_DIS
LIN {X 0.108,Y -425.975,Z 594.578,A 0.000,B 0.000,C 90.000,E1 104.064} C_DIS
LIN {X 0.173,Y -445.853,Z 594.567,A 0.000,B 0.000,C 90.000,E1 101.951} C_DIS
LIN {X 0.176,Y -466.338,Z 594.556,A 0.000,B 0.000,C 90.000,E1 100.018} C_DIS
LIN {X -0.165,Y -473.965,Z 594.552,A 0.000,B 0.000,C 90.000,E1 99.378} C_DIS
LIN {X -0.148,Y -475.816,Z 594.551,A 0.000,B 0.000,C 90.000,E1 99.151} C_DIS
LIN {X 0.186,Y -477.396,Z 594.549,A 0.000,B 0.000,C 90.000,E1 98.859} C_DIS
LIN {X 0.048,Y -478.581,Z 594.548,A 0.000,B 0.000,C 90.000,E1 98.624} C_DIS
LIN {X 0.192,Y -480.020,Z 594.545,A 0.000,B 0.000,C 90.000,E1 98.106} C_DIS
LIN {X -0.131,Y -480.424,Z 594.542,A 0.000,B 0.000,C 90.000,E1 97.644} C_DIS
LIN {X 0.032,Y -479.857,Z 594.540,A 0.000,B 0.000,C 90.000,E1 97.125} C_DIS
LIN {X 0.198,Y -478.230,Z 594.537,A 0.000,B 0.000,C 90.000,E1 96.606} C_DIS
LIN {X 0.068,Y -476.930,Z 594.535,A 0.000,B 0.000,C 90.000,E1 96.372} C_DIS
LIN {X 0.030,Y -471.437,Z 594.531,A 0.000,B 0.000,C 90.000,E1 95.625} C_DIS
LIN {X 0.097,Y -458.745,Z 594.521,A 0.000,B 0.000,C 90.000,E1 93.841} C_DIS
LIN {X -0.134,Y -447.518,Z 594.511,A 0.000,B 0.000,C 90.000,E1 92.064} C_DIS
LIN {X 0.037,Y -435.910,Z 594.500,A 0.000,B 0.000,C 90.000,E1 89.943} C_DIS
LIN {X -0.058,Y -428.399,Z 594.492,A 0.000,B 0.000,C 90.000,E1 88.625} C_DIS
LIN {X -0.134,Y -418.983,Z 594.483,A 0.000,B 0.000,C 90.000,E1 87.020} C_DIS
LIN {X -0.015,Y -403.232,Z 594.468,A 0.000,B 0.000,C 90.000,E1 84.261} C_DIS
LIN {X 0.071,Y -389.805,Z 594.454,A 0.000,B 0.000,C 90.000,E1 81.724} C_DIS
LIN {X -0.032,Y -376.709,Z 594.440,A 0.000,B 0.000,C 90.000,E1 79.162} C_DIS
LIN {X 0.045,Y -364.062,Z 594.425,A 0.000,B 0.000,C 90.000,E1 76.520} C_DIS
LIN {X -0.177,Y -349.411,Z 594.407,A 0.000,B 0.000,C 90.000,E1 73.268} C_DIS
LIN {X -0.044,Y -335.170,Z 594.386,A 0.000,B 0.000,C 90.000,E1 69.571} C_DIS
LIN {X 0.070,Y -325.667,Z 594.371,A 0.000,B 0.000,C 90.000,E1 66.741} C_DIS
LIN {X -0.046,Y -315.879,Z 594.353,A 0.000,B 0.000,C 90.000,E1 63.589} C_DIS
LIN {X 0.010,Y -308.440,Z 594.339,A 0.000,B 0.000,C 90.000,E1 61.001} C_DIS
LIN {X -0.085,Y -301.163,Z 594.324,A 0.000,B 0.000,C 90.000,E1 58.408} C_DIS
LIN {X -0.116,Y -292.537,Z 594.306,A 0.000,B 0.000,C 90.000,E1 55.102} C_DIS
LIN {X -0.022,Y -285.964,Z 594.291,A 0.000,B 0.000,C 90.000,E1 52.396} C_DIS
LIN {X -0.003,Y -280.983,Z 594.280,A 0.000,B 0.000,C 90.000,E1 50.356} C_DIS
LIN {X -0.116,Y -275.659,Z 594.268,A 0.000,B 0.000,C 90.000,E1 48.324} C_DIS
LIN {X 0.059,Y -271.808,Z 594.261,A 0.000,B 0.000,C 90.000,E1 46.905} C_DIS
LIN {X 0.063,Y -266.528,Z 594.251,A 0.000,B 0.000,C 90.000,E1 45.162} C_DIS
LIN {X 0.015,Y -259.730,Z 594.239,A 0.000,B 0.000,C 90.000,E1 43.056} C_DIS
LIN {X 0.084,Y -250.621,Z 594.223,A 0.000,B 0.000,C 90.000,E1 40.172} C_DIS
LIN {X -0.031,Y -240.955,Z 594.205,A 0.000,B 0.000,C 90.000,E1 36.916} C_DIS
LIN {X 0.109,Y -233.203,Z 594.189,A 0.000,B 0.000,C 90.000,E1 33.913} C_DIS
LIN {X -0.002,Y -226.174,Z 594.172,A 0.000,B 0.000,C 90.000,E1 30.924} C_DIS
LIN {X 0.070,Y -219.785,Z 594.155,A 0.000,B 0.000,C 90.000,E1 27.847} C_DIS
LIN {X 0.124,Y -212.904,Z 594.133,A 0.000,B 0.000,C 90.000,E1 23.951} C_DIS
LIN {X -0.017,Y -208.297,Z 594.116,A 0.000,B 0.000,C 90.000,E1 20.844} C_DIS
LIN {X 0.027,Y -203.601,Z 594.094,A 0.000,B 0.000,C 90.000,E1 16.858} C_DIS
LIN {X -0.053,Y -199.404,Z 594.067,A 0.000,B 0.000,C 90.000,E1 12.063} C_DIS
LIN {X 0.011,Y -196.437,Z 594.035,A 0.000,B 0.000,C 90.000,E1 6.372} C_DIS
LIN {X 0.067,Y -197.647,Z 593.961,A 0.000,B 0.000,C 90.000,E1 352.996} C_DIS
LIN {X -0.072,Y -200.828,Z 593.934,A 0.000,B 0.000,C 90.000,E1 348.173} C_DIS
LIN {X 0.017,Y -205.234,Z 593.907,A 0.000,B 0.000,C 90.000,E1 343.323} C_DIS
LIN {X 0.026,Y -209.817,Z 593.885,A 0.000,B 0.000,C 90.000,E1 339.337} C_DIS
LIN {X -0.031,Y -215.201,Z 593.863,A 0.000,B 0.000,C 90.000,E1 335.409} C_DIS
LIN {X -0.036,Y -221.246,Z 593.842,A 0.000,B 0.000,C 90.000,E1 331.513} C_DIS
LIN {X -0.013,Y -227.942,Z 593.820,A 0.000,B 0.000,C 90.000,E1 327.661} C_DIS
LIN {X 0.042,Y -233.635,Z 593.803,A 0.000,B 0.000,C 90.000,E1 324.609} C_DIS
LIN {X -0.053,Y -241.099,Z 593.783,A 0.000,B 0.000,C 90.000,E1 320.884} C_DIS
LIN {X -0.026,Y -249.299,Z 593.762,A 0.000,B 0.000,C 90.000,E1 317.187} C_DIS
LIN {X 0.046,Y -258.493,Z 593.742,A 0.000,B 0.000,C 90.000,E1 313.542} C_DIS
LIN {X -0.008,Y -266.790,Z 593.726,A 0.000,B 0.000,C 90.000,E1 310.701} C_DIS
LIN {X 0.026,Y -276.281,Z 593.711,A 0.000,B 0.000,C 90.000,E1 307.890} C_DIS
LIN {X -0.074,Y -288.131,Z 593.693,A 0.000,B 0.000,C 90.000,E1 304.818} C_DIS
LIN {X -0.104,Y -299.836,Z 593.678,A 0.000,B 0.000,C 90.000,E1 302.133} C_DIS
LIN {X 0.055,Y -315.661,Z 593.660,A 0.000,B 0.000,C 90.000,E1 298.821} C_DIS
LIN {X -0.015,Y -332.443,Z 593.642,A 0.000,B 0.000,C 90.000,E1 295.643} C_DIS
LIN {X 0.000,Y -345.195,Z 593.630,A 0.000,B 0.000,C 90.000,E1 293.462} C_DIS
LIN {X -0.037,Y -363.104,Z 593.615,A 0.000,B 0.000,C 90.000,E1 290.737} C_DIS
LIN {X 0.175,Y -382.983,Z 593.600,A 0.000,B 0.000,C 90.000,E1 288.055} C_DIS
LIN {X -0.009,Y -399.363,Z 593.589,A 0.000,B 0.000,C 90.000,E1 286.079} C_DIS
LIN {X -0.078,Y -413.362,Z 593.580,A 0.000,B 0.000,C 90.000,E1 284.411} C_DIS
LIN {X -0.098,Y -427.235,Z 593.571,A 0.000,B 0.000,C 90.000,E1 282.771} C_DIS
LIN {X 0.178,Y -436.020,Z 593.565,A 0.000,B 0.000,C 90.000,E1 281.658} C_DIS
LIN {X -0.086,Y -446.391,Z 593.558,A 0.000,B 0.000,C 90.000,E1 280.366} C_DIS
LIN {X -0.101,Y -454.193,Z 593.552,A 0.000,B 0.000,C 90.000,E1 279.321} C_DIS
LIN {X -0.024,Y -461.391,Z 593.546,A 0.000,B 0.000,C 90.000,E1 278.276} C_DIS
LIN {X 0.077,Y -468.041,Z 593.540,A 0.000,B 0.000,C 90.000,E1 277.239} C_DIS
LIN {X -0.210,Y -474.058,Z 593.535,A 0.000,B 0.000,C 90.000,E1 276.258} C_DIS
LIN {X 0.191,Y -477.975,Z 593.530,A 0.000,B 0.000,C 90.000,E1 275.454} C_DIS
LIN {X 0.192,Y -481.134,Z 593.526,A 0.000,B 0.000,C 90.000,E1 274.702} C_DIS
LIN {X -0.170,Y -482.801,Z 593.523,A 0.000,B 0.000,C 90.000,E1 274.245} C_DIS
LIN {X -0.004,Y -484.158,Z 593.521,A 0.000,B 0.000,C 90.000,E1 273.726} C_DIS
LIN {X 0.143,Y -485.160,Z 593.518,A 0.000,B 0.000,C 90.000,E1 273.212} C_DIS
LIN {X -0.161,Y -485.925,Z 593.515,A 0.000,B 0.000,C 90.000,E1 272.751} C_DIS
LIN {X 0.002,Y -486.369,Z 593.512,A 0.000,B 0.000,C 90.000,E1 272.236} C_DIS
LIN {X 0.187,Y -486.443,Z 593.510,A 0.000,B 0.000,C 90.000,E1 271.718} C_DIS
LIN {X -0.128,Y -486.109,Z 593.507,A 0.000,B 0.000,C 90.000,E1 271.260} C_DIS
LIN {X 0.045,Y -485.321,Z 593.504,A 0.000,B 0.000,C 90.000,E1 270.745} C_DIS
LIN {X 0.216,Y -483.977,Z 593.501,A 0.000,B 0.000,C 90.000,E1 270.229} C_DIS
LIN {X -0.100,Y -482.053,Z 593.499,A 0.000,B 0.000,C 90.000,E1 269.771} C_DIS
LIN {X 0.058,Y -479.364,Z 593.496,A 0.000,B 0.000,C 90.000,E1 269.255} C_DIS
LIN {X 0.196,Y -475.795,Z 593.493,A 0.000,B 0.000,C 90.000,E1 268.740} C_DIS
LIN {X -0.159,Y -471.177,Z 593.490,A 0.000,B 0.000,C 90.000,E1 268.282} C_DIS
LIN {X 0.145,Y -468.467,Z 593.489,A 0.000,B 0.000,C 90.000,E1 267.993} C_DIS
LIN {X -0.036,Y -465.362,Z 593.488,A 0.000,B 0.000,C 90.000,E1 267.764} C_DIS
LIN {X 0.173,Y -458.955,Z 593.485,A 0.000,B 0.000,C 90.000,E1 267.306} C_DIS
LIN {X 0.002,Y -451.953,Z 593.483,A 0.000,B 0.000,C 90.000,E1 266.963} C_DIS
LIN {X -0.023,Y -444.499,Z 593.482,A 0.000,B 0.000,C 90.000,E1 266.674} C_DIS
LIN {X -0.004,Y -436.754,Z 593.480,A 0.000,B 0.000,C 90.000,E1 266.445} C_DIS
LIN {X 0.025,Y -428.499,Z 593.479,A 0.000,B 0.000,C 90.000,E1 266.274} C_DIS
LIN {X -0.001,Y -418.900,Z 593.479,A 0.000,B 0.000,C 90.000,E1 266.159} C_DIS
LIN {X -0.024,Y -408.523,Z 593.478,A 0.000,B 0.000,C 90.000,E1 266.102} C_DIS
LIN {X -0.042,Y -180.924,Z 593.478,A 0.000,B 0.000,C 90.000,E1 266.102} C_DIS
LIN {X 0.002,Y -180.875,Z 593.473,A 0.000,B 0.000,C 90.000,E1 265.065} C_DIS
LIN {X 0.085,Y -178.942,Z 593.443,A 0.000,B 0.000,C 90.000,E1 259.803} C_DIS
LIN {X -0.048,Y -175.992,Z 593.415,A 0.000,B 0.000,C 90.000,E1 254.755} C_DIS
LIN {X 0.067,Y -175.495,Z 593.410,A 0.000,B 0.000,C 90.000,E1 253.866} C_DIS
LIN {X -0.039,Y -172.238,Z 593.387,A 0.000,B 0.000,C 90.000,E1 249.625} C_DIS
LIN {X -0.060,Y -171.715,Z 593.382,A 0.000,B 0.000,C 90.000,E1 248.773} C_DIS
LIN {X 0.024,Y -167.310,Z 593.353,A 0.000,B 0.000,C 90.000,E1 243.563} C_DIS
LIN {X 0.030,Y -166.691,Z 593.348,A 0.000,B 0.000,C 90.000,E1 242.692} C_DIS
LIN {X 0.020,Y -162.672,Z 593.324,A 0.000,B 0.000,C 90.000,E1 238.329} C_DIS
LIN {X -0.006,Y -161.362,Z 593.314,A 0.000,B 0.000,C 90.000,E1 236.580} C_DIS
LIN {X 0.027,Y -157.356,Z 593.290,A 0.000,B 0.000,C 90.000,E1 232.145} C_DIS
LIN {X 0.056,Y -155.344,Z 593.275,A 0.000,B 0.000,C 90.000,E1 229.461} C_DIS
LIN {X -0.014,Y -151.691,Z 593.250,A 0.000,B 0.000,C 90.000,E1 225.000} C_DIS
LIN {X 0.034,Y -150.554,Z 593.240,A 0.000,B 0.000,C 90.000,E1 223.176} C_DIS
LIN {X -0.049,Y -147.280,Z 593.215,A 0.000,B 0.000,C 90.000,E1 218.669} C_DIS
LIN {X 0.038,Y -145.309,Z 593.194,A 0.000,B 0.000,C 90.000,E1 214.978} C_DIS
LIN {X 0.030,Y -142.399,Z 593.164,A 0.000,B 0.000,C 90.000,E1 209.461} C_DIS
LIN {X 0.013,Y -141.381,Z 593.148,A 0.000,B 0.000,C 90.000,E1 206.693} C_DIS
LIN {X 0.054,Y -139.349,Z 593.112,A 0.000,B 0.000,C 90.000,E1 200.174} C_DIS
LIN {X -0.004,Y -138.786,Z 593.097,A 0.000,B 0.000,C 90.000,E1 197.402} C_DIS
LIN {X 0.054,Y -138.344,Z 593.055,A 0.000,B 0.000,C 90.000,E1 189.905} C_DIS
LIN {X -0.065,Y -139.387,Z 593.008,A 0.000,B 0.000,C 90.000,E1 181.547} C_DIS
LIN {X -0.012,Y -141.283,Z 592.972,A 0.000,B 0.000,C 90.000,E1 175.008} C_DIS
LIN {X -0.054,Y -142.647,Z 592.957,A 0.000,B 0.000,C 90.000,E1 172.243} C_DIS
LIN {X 0.037,Y -144.983,Z 592.931,A 0.000,B 0.000,C 90.000,E1 167.589} C_DIS
LIN {X 0.028,Y -147.611,Z 592.911,A 0.000,B 0.000,C 90.000,E1 163.921} C_DIS
LIN {X -0.034,Y -150.233,Z 592.890,A 0.000,B 0.000,C 90.000,E1 160.296} C_DIS
LIN {X -0.019,Y -153.624,Z 592.870,A 0.000,B 0.000,C 90.000,E1 156.666} C_DIS
LIN {X -0.031,Y -157.040,Z 592.850,A 0.000,B 0.000,C 90.000,E1 153.076} C_DIS
LIN {X 0.038,Y -161.165,Z 592.831,A 0.000,B 0.000,C 90.000,E1 149.488} C_DIS
LIN {X -0.018,Y -163.261,Z 592.821,A 0.000,B 0.000,C 90.000,E1 147.740} C_DIS
LIN {X 0.080,Y -167.701,Z 592.801,A 0.000,B 0.000,C 90.000,E1 144.196} C_DIS
LIN {X -0.007,Y -171.521,Z 592.787,A 0.000,B 0.000,C 90.000,E1 141.618} C_DIS
LIN {X 0.037,Y -176.459,Z 592.768,A 0.000,B 0.000,C 90.000,E1 138.162} C_DIS
LIN {X -0.094,Y -180.755,Z 592.753,A 0.000,B 0.000,C 90.000,E1 135.648} C_DIS
LIN {X 0.024,Y -186.161,Z 592.735,A 0.000,B 0.000,C 90.000,E1 132.243} C_DIS
LIN {X 0.015,Y -191.369,Z 592.719,A 0.000,B 0.000,C 90.000,E1 129.402} C_DIS
LIN {X -0.013,Y -288.895,Z 592.719,A 0.000,B 0.000,C 90.000,E1 129.402} C_DIS
LIN {X -0.071,Y -291.304,Z 592.719,A 0.000,B 0.000,C 90.000,E1 129.358} C_DIS
LIN {X 0.094,Y -295.123,Z 592.717,A 0.000,B 0.000,C 90.000,E1 129.116} C_DIS
LIN {X 0.073,Y -297.452,Z 592.716,A 0.000,B 0.000,C 90.000,E1 128.910} C_DIS
LIN {X 0.105,Y -301.282,Z 592.713,A 0.000,B 0.000,C 90.000,E1 128.382} C_DIS
LIN {X -0.138,Y -302.974,Z 592.711,A 0.000,B 0.000,C 90.000,E1 128.096} C_DIS
LIN {X 0.045,Y -304.302,Z 592.710,A 0.000,B 0.000,C 90.000,E1 127.729} C_DIS
LIN {X -0.148,Y -312.927,Z 592.693,A 0.000,B 0.000,C 90.000,E1 124.818} C_DIS
LIN {X -0.098,Y -323.762,Z 592.675,A 0.000,B 0.000,C 90.000,E1 121.592} C_DIS
LIN {X -0.051,Y -334.896,Z 592.660,A 0.000,B 0.000,C 90.000,E1 118.743} C_DIS
LIN {X -0.160,Y -347.439,Z 592.644,A 0.000,B 0.000,C 90.000,E1 115.976} C_DIS
LIN {X 0.056,Y -359.867,Z 592.631,A 0.000,B 0.000,C 90.000,E1 113.515} C_DIS
LIN {X -0.032,Y -373.589,Z 592.617,A 0.000,B 0.000,C 90.000,E1 111.153} C_DIS
LIN {X -0.058,Y -388.704,Z 592.605,A 0.000,B 0.000,C 90.000,E1 108.833} C_DIS
LIN {X 0.044,Y -405.322,Z 592.592,A 0.000,B 0.000,C 90.000,E1 106.551} C_DIS
LIN {X -0.056,Y -423.566,Z 592.580,A 0.000,B 0.000,C 90.000,E1 104.356} C_DIS
LIN {X -0.135,Y -443.314,Z 592.568,A 0.000,B 0.000,C 90.000,E1 102.243} C_DIS
LIN {X 0.140,Y -463.733,Z 592.557,A 0.000,B 0.000,C 90.000,E1 100.254} C_DIS
LIN {X -0.186,Y -473.985,Z 592.552,A 0.000,B 0.000,C 90.000,E1 99.378} C_DIS
LIN {X -0.169,Y -475.859,Z 592.551,A 0.000,B 0.000,C 90.000,E1 99.151} C_DIS
LIN {X 0.165,Y -477.459,Z 592.549,A 0.000,B 0.000,C 90.000,E1 98.859} C_DIS
LIN {X 0.027,Y -478.658,Z 592.548,A 0.000,B 0.000,C 90.000,E1 98.624} C_DIS
LIN {X 0.172,Y -480.117,Z 592.545,A 0.000,B 0.000,C 90.000,E1 98.106} C_DIS
LIN {X -0.150,Y -480.537,Z 592.542,A 0.000,B 0.000,C 90.000,E1 97.644} C_DIS
LIN {X 0.013,Y -479.988,Z 592.540,A 0.000,B 0.000,C 90.000,E1 97.125} C_DIS
LIN {X 0.179,Y -478.383,Z 592.537,A 0.000,B 0.000,C 90.000,E1 96.606} C_DIS
LIN {X 0.049,Y -477.096,Z 592.535,A 0.000,B 0.000,C 90.000,E1 96.372} C_DIS
LIN {X 0.012,Y -471.614,Z 592.531,A 0.000,B 0.000,C 90.000,E1 95.625} C_DIS
LIN {X 0.083,Y -458.900,Z 592.521,A 0.000,B 0.000,C 90.000,E1 93.841} C_DIS
LIN {X -0.144,Y -447.623,Z 592.511,A 0.000,B 0.000,C 90.000,E1 92.064} C_DIS
LIN {X 0.030,Y -436.010,Z 592.500,A 0.000,B 0.000,C 90.000,E1 89.943} C_DIS
LIN {X -0.064,Y -428.487,Z 592.492,A 0.000,B 0.000,C 90.000,E1 88.625} C_DIS
LIN {X 0.171,Y -420.650,Z 592.485,A 0.000,B 0.000,C 90.000,E1 87.249} C_DIS
LIN {X -0.173,Y -406.369,Z 592.471,A 0.000,B 0.000,C 90.000,E1 84.837} C_DIS
LIN {X 0.066,Y -391.339,Z 592.456,A 0.000,B 0.000,C 90.000,E1 82.008} C_DIS
LIN {X -0.079,Y -379.626,Z 592.443,A 0.000,B 0.000,C 90.000,E1 79.746} C_DIS
LIN {X -0.004,Y -366.836,Z 592.428,A 0.000,B 0.000,C 90.000,E1 77.117} C_DIS
LIN {X -0.105,Y -350.671,Z 592.409,A 0.000,B 0.000,C 90.000,E1 73.559} C_DIS
LIN {X -0.043,Y -335.188,Z 592.386,A 0.000,B 0.000,C 90.000,E1 69.571} C_DIS
LIN {X 0.124,Y -323.702,Z 592.367,A 0.000,B 0.000,C 90.000,E1 66.102} C_DIS
LIN {X -0.046,Y -314.058,Z 592.350,A 0.000,B 0.000,C 90.000,E1 62.948} C_DIS
LIN {X 0.111,Y -306.670,Z 592.335,A 0.000,B 0.000,C 90.000,E1 60.333} C_DIS
LIN {X -0.027,Y -299.480,Z 592.321,A 0.000,B 0.000,C 90.000,E1 57.740} C_DIS
LIN {X 0.050,Y -290.911,Z 592.302,A 0.000,B 0.000,C 90.000,E1 54.402} C_DIS
LIN {X 0.095,Y -284.378,Z 592.287,A 0.000,B 0.000,C 90.000,E1 51.698} C_DIS
LIN {X 0.040,Y -279.292,Z 592.276,A 0.000,B 0.000,C 90.000,E1 49.666} C_DIS
LIN {X -0.105,Y -273.789,Z 592.265,A 0.000,B 0.000,C 90.000,E1 47.634} C_DIS
LIN {X 0.046,Y -269.759,Z 592.257,A 0.000,B 0.000,C 90.000,E1 46.215} C_DIS
LIN {X 0.014,Y -264.289,Z 592.247,A 0.000,B 0.000,C 90.000,E1 44.474} C_DIS
LIN {X -0.028,Y -256.283,Z 592.233,A 0.000,B 0.000,C 90.000,E1 42.000} C_DIS
LIN {X -0.022,Y -245.111,Z 592.213,A 0.000,B 0.000,C 90.000,E1 38.382} C_DIS
LIN {X -0.019,Y -236.955,Z 592.197,A 0.000,B 0.000,C 90.000,E1 35.438} C_DIS
LIN {X 0.089,Y -229.560,Z 592.180,A 0.000,B 0.000,C 90.000,E1 32.418} C_DIS
LIN {X -0.031,Y -222.856,Z 592.163,A 0.000,B 0.000,C 90.000,E1 29.411} C_DIS
LIN {X 0.053,Y -216.878,Z 592.146,A 0.000,B 0.000,C 90.000,E1 26.309} C_DIS
LIN {X -0.007,Y -211.630,Z 592.129,A 0.000,B 0.000,C 90.000,E1 23.206} C_DIS
LIN {X -0.038,Y -206.261,Z 592.107,A 0.000,B 0.000,C 90.000,E1 19.268} C_DIS
LIN {X 0.079,Y -202.014,Z 592.085,A 0.000,B 0.000,C 90.000,E1 15.245} C_DIS
LIN {X 0.001,Y -198.297,Z 592.058,A 0.000,B 0.000,C 90.000,E1 10.433} C_DIS
LIN {X -0.069,Y -195.792,Z 592.022,A 0.000,B 0.000,C 90.000,E1 3.955} C_DIS
LIN {X 0.101,Y -197.273,Z 591.966,A 0.000,B 0.000,C 90.000,E1 353.799} C_DIS
LIN {X -0.074,Y -200.189,Z 591.939,A 0.000,B 0.000,C 90.000,E1 348.982} C_DIS
LIN {X -0.100,Y -204.450,Z 591.912,A 0.000,B 0.000,C 90.000,E1 344.157} C_DIS
LIN {X 0.013,Y -208.852,Z 591.890,A 0.000,B 0.000,C 90.000,E1 340.134} C_DIS
LIN {X 0.035,Y -214.073,Z 591.868,A 0.000,B 0.000,C 90.000,E1 336.177} C_DIS
LIN {X -0.005,Y -220.007,Z 591.846,A 0.000,B 0.000,C 90.000,E1 332.281} C_DIS
LIN {X 0.063,Y -226.577,Z 591.825,A 0.000,B 0.000,C 90.000,E1 328.408} C_DIS
LIN {X -0.048,Y -232.209,Z 591.808,A 0.000,B 0.000,C 90.000,E1 325.388} C_DIS
LIN {X -0.001,Y -239.539,Z 591.787,A 0.000,B 0.000,C 90.000,E1 321.618} C_DIS
LIN {X -0.017,Y -247.561,Z 591.766,A 0.000,B 0.000,C 90.000,E1 317.919} C_DIS
LIN {X 0.011,Y -256.526,Z 591.746,A 0.000,B 0.000,C 90.000,E1 314.271} C_DIS
LIN {X -0.006,Y -266.741,Z 591.726,A 0.000,B 0.000,C 90.000,E1 310.701} C_DIS
LIN {X 0.028,Y -276.217,Z 591.711,A 0.000,B 0.000,C 90.000,E1 307.890} C_DIS
LIN {X -0.107,Y -289.487,Z 591.691,A 0.000,B 0.000,C 90.000,E1 304.485} C_DIS
LIN {X -0.069,Y -304.384,Z 591.673,A 0.000,B 0.000,C 90.000,E1 301.131} C_DIS
LIN {X 0.107,Y -317.191,Z 591.658,A 0.000,B 0.000,C 90.000,E1 298.487} C_DIS
LIN {X -0.061,Y -334.102,Z 591.641,A 0.000,B 0.000,C 90.000,E1 295.335} C_DIS
LIN {X 0.146,Y -348.932,Z 591.627,A 0.000,B 0.000,C 90.000,E1 292.823} C_DIS
LIN {X 0.084,Y -367.305,Z 591.612,A 0.000,B 0.000,C 90.000,E1 290.120} C_DIS
LIN {X -0.070,Y -387.557,Z 591.597,A 0.000,B 0.000,C 90.000,E1 287.511} C_DIS
LIN {X 0.034,Y -401.727,Z 591.588,A 0.000,B 0.000,C 90.000,E1 285.788} C_DIS
LIN {X 0.014,Y -415.716,Z 591.578,A 0.000,B 0.000,C 90.000,E1 284.120} C_DIS
LIN {X -0.115,Y -427.292,Z 591.571,A 0.000,B 0.000,C 90.000,E1 282.771} C_DIS
LIN {X 0.161,Y -436.093,Z 591.565,A 0.000,B 0.000,C 90.000,E1 281.658} C_DIS
LIN {X 0.116,Y -444.400,Z 591.559,A 0.000,B 0.000,C 90.000,E1 280.602} C_DIS
LIN {X -0.117,Y -454.237,Z 591.552,A 0.000,B 0.000,C 90.000,E1 279.321} C_DIS
LIN {X -0.039,Y -461.422,Z 591.546,A 0.000,B 0.000,C 90.000,E1 278.276} C_DIS
LIN {X 0.060,Y -468.065,Z 591.540,A 0.000,B 0.000,C 90.000,E1 277.239} C_DIS
LIN {X -0.224,Y -474.064,Z 591.535,A 0.000,B 0.000,C 90.000,E1 276.258} C_DIS
LIN {X 0.176,Y -477.975,Z 591.530,A 0.000,B 0.000,C 90.000,E1 275.454} C_DIS
LIN {X 0.177,Y -481.102,Z 591.526,A 0.000,B 0.000,C 90.000,E1 274.702} C_DIS
LIN {X -0.186,Y -482.807,Z 591.523,A 0.000,B 0.000,C 90.000,E1 274.245} C_DIS
LIN {X -0.020,Y -484.163,Z 591.521,A 0.000,B 0.000,C 90.000,E1 273.726} C_DIS
LIN {X 0.127,Y -485.212,Z 591.518,A 0.000,B 0.000,C 90.000,E1 273.212} C_DIS
LIN {X -0.178,Y -485.977,Z 591.515,A 0.000,B 0.000,C 90.000,E1 272.751} C_DIS
LIN {X -0.014,Y -486.421,Z 591.512,A 0.000,B 0.000,C 90.000,E1 272.236} C_DIS
LIN {X 0.171,Y -486.515,Z 591.510,A 0.000,B 0.000,C 90.000,E1 271.718} C_DIS
LIN {X -0.143,Y -486.148,Z 591.507,A 0.000,B 0.000,C 90.000,E1 271.260} C_DIS
LIN {X 0.030,Y -485.346,Z 591.504,A 0.000,B 0.000,C 90.000,E1 270.745} C_DIS
LIN {X 0.202,Y -484.019,Z 591.501,A 0.000,B 0.000,C 90.000,E1 270.229} C_DIS
LIN {X -0.114,Y -482.058,Z 591.499,A 0.000,B 0.000,C 90.000,E1 269.771} C_DIS
LIN {X 0.045,Y -479.348,Z 591.496,A 0.000,B 0.000,C 90.000,E1 269.255} C_DIS
LIN {X -0.125,Y -477.708,Z 591.495,A 0.000,B 0.000,C 90.000,E1 269.026} C_DIS
LIN {X 0.004,Y -473.633,Z 591.492,A 0.000,B 0.000,C 90.000,E1 268.511} C_DIS
LIN {X 0.140,Y -468.447,Z 591.489,A 0.000,B 0.000,C 90.000,E1 267.993} C_DIS
LIN {X 0.075,Y -462.373,Z 591.486,A 0.000,B 0.000,C 90.000,E1 267.535} C_DIS
LIN {X 0.178,Y -458.990,Z 591.485,A 0.000,B 0.000,C 90.000,E1 267.306} C_DIS
LIN {X 0.017,Y -451.880,Z 591.483,A 0.000,B 0.000,C 90.000,E1 266.963} C_DIS
LIN {X 0.042,Y -444.757,Z 591.482,A 0.000,B 0.000,C 90.000,E1 266.674} C_DIS
LIN {X 0.058,Y -437.137,Z 591.480,A 0.000,B 0.000,C 90.000,E1 266.445} C_DIS
LIN {X 0.047,Y -428.742,Z 591.479,A 0.000,B 0.000,C 90.000,E1 266.274} C_DIS
LIN {X 0.007,Y -419.086,Z 591.479,A 0.000,B 0.000,C 90.000,E1 266.159} C_DIS
LIN {X -0.022,Y -409.703,Z 591.478,A 0.000,B 0.000,C 90.000,E1 266.102} C_DIS
LIN {X -0.095,Y -405.943,Z 591.478,A 0.000,B 0.000,C 90.000,E1 266.102} C_DIS
LIN {X -0.074,Y -180.924,Z 591.478,A 0.000,B 0.000,C 90.000,E1 266.102} C_DIS
LIN {X -0.028,Y -180.874,Z 591.473,A 0.000,B 0.000,C 90.000,E1 265.065} C_DIS
LIN {X 0.053,Y -178.938,Z 591.443,A 0.000,B 0.000,C 90.000,E1 259.803} C_DIS
LIN {X -0.078,Y -175.988,Z 591.415,A 0.000,B 0.000,C 90.000,E1 254.755} C_DIS
LIN {X 0.036,Y -175.487,Z 591.410,A 0.000,B 0.000,C 90.000,E1 253.866} C_DIS
LIN {X 0.092,Y -172.231,Z 591.387,A 0.000,B 0.000,C 90.000,E1 249.571} C_DIS
LIN {X 0.070,Y -171.708,Z 591.382,A 0.000,B 0.000,C 90.000,E1 248.720} C_DIS
LIN {X -0.005,Y -167.303,Z 591.353,A 0.000,B 0.000,C 90.000,E1 243.563} C_DIS
